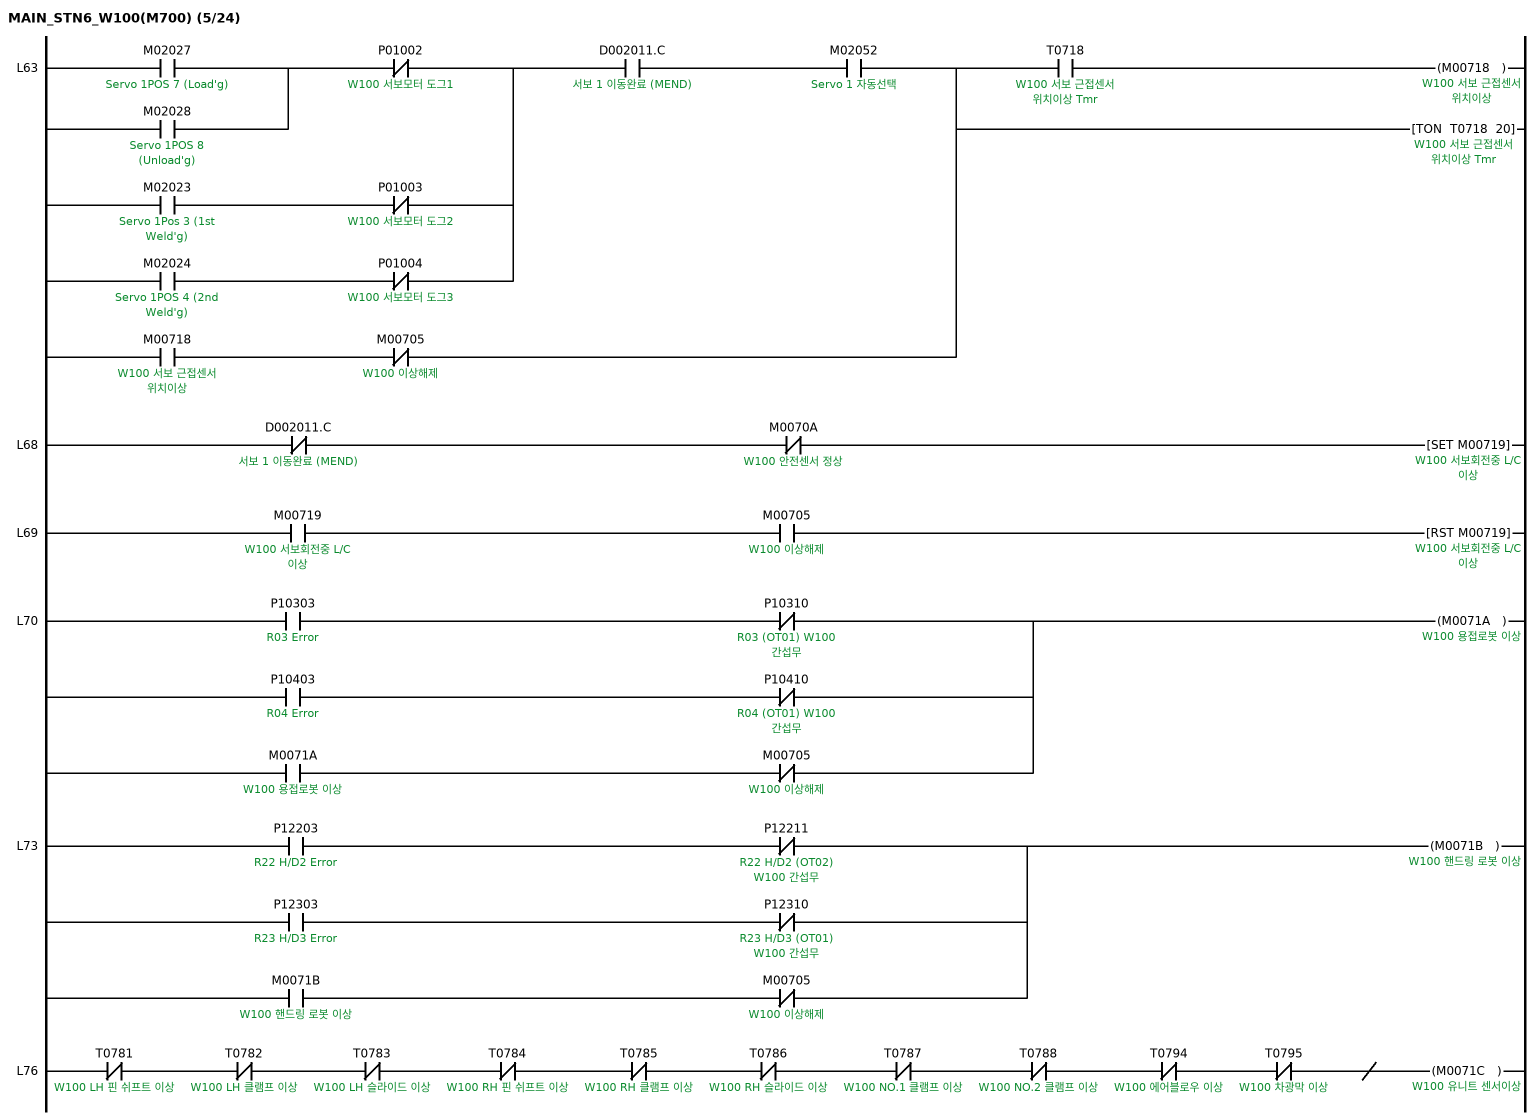
[picture p120: MAIN_STN6_W100(M700) rungs L63-L76]
; L63
LOAD      M02027	// Servo 1POS 7 (Load'g)
OR        M02028	// Servo 1POS 8 (Unload'g)
AND NOT   P01002	// W100 서보모터 도그1
LOAD      M02023	// Servo 1Pos 3 (1st Weld'g)
AND NOT   P01003	// W100 서보모터 도그2
OR LOAD
LOAD      M02024	// Servo 1POS 4 (2nd Weld'g)
AND NOT   P01004	// W100 서보모터 도그3
OR LOAD
AND       D002011.C	// 서보 1 이동완료 (MEND)
AND       M02052	// Servo 1 자동선택
LOAD      M00718	// W100 서보 근접센서 위치이상
AND NOT   M00705	// W100 이상해제
OR LOAD
MPUSH
AND       T0718	// W100 서보 근접센서 위치이상 Tmr
OUT       M00718	// W100 서보 근접센서 위치이상
MPOP
TON       T0718 20	// W100 서보 근접센서 위치이상 Tmr
; L68
LOAD NOT  D002011.C	// 서보 1 이동완료 (MEND)
AND NOT   M0070A	// W100 안전센서 정상
SET       M00719	// W100 서보회전중 L/C 이상
; L69
LOAD      M00719	// W100 서보회전중 L/C 이상
AND       M00705	// W100 이상해제
RST       M00719	// W100 서보회전중 L/C 이상
; L70
LOAD      P10303	// R03 Error
AND NOT   P10310	// R03 (OT01) W100 간섭무
LOAD      P10403	// R04 Error
AND NOT   P10410	// R04 (OT01) W100 간섭무
OR LOAD
LOAD      M0071A	// W100 용접로봇 이상
AND NOT   M00705	// W100 이상해제
OR LOAD
OUT       M0071A	// W100 용접로봇 이상
; L73
LOAD      P12203	// R22 H/D2 Error
AND NOT   P12211	// R22 H/D2 (OT02) W100 간섭무
LOAD      P12303	// R23 H/D3 Error
AND NOT   P12310	// R23 H/D3 (OT01) W100 간섭무
OR LOAD
LOAD      M0071B	// W100 핸드링 로봇 이상
AND NOT   M00705	// W100 이상해제
OR LOAD
OUT       M0071B	// W100 핸드링 로봇 이상
; L76
LOAD NOT  T0781	// W100 LH 핀 쉬프트 이상
AND NOT   T0782	// W100 LH 클램프 이상
AND NOT   T0783	// W100 LH 슬라이드 이상
AND NOT   T0784	// W100 RH 핀 쉬프트 이상
AND NOT   T0785	// W100 RH 클램프 이상
AND NOT   T0786	// W100 RH 슬라이드 이상
AND NOT   T0787	// W100 NO.1 클램프 이상
AND NOT   T0788	// W100 NO.2 클램프 이상
AND NOT   T0794	// W100 에어블로우 이상
AND NOT   T0795	// W100 차광막 이상
NOT
OUT       M0071C	// W100 유니트 센서이상

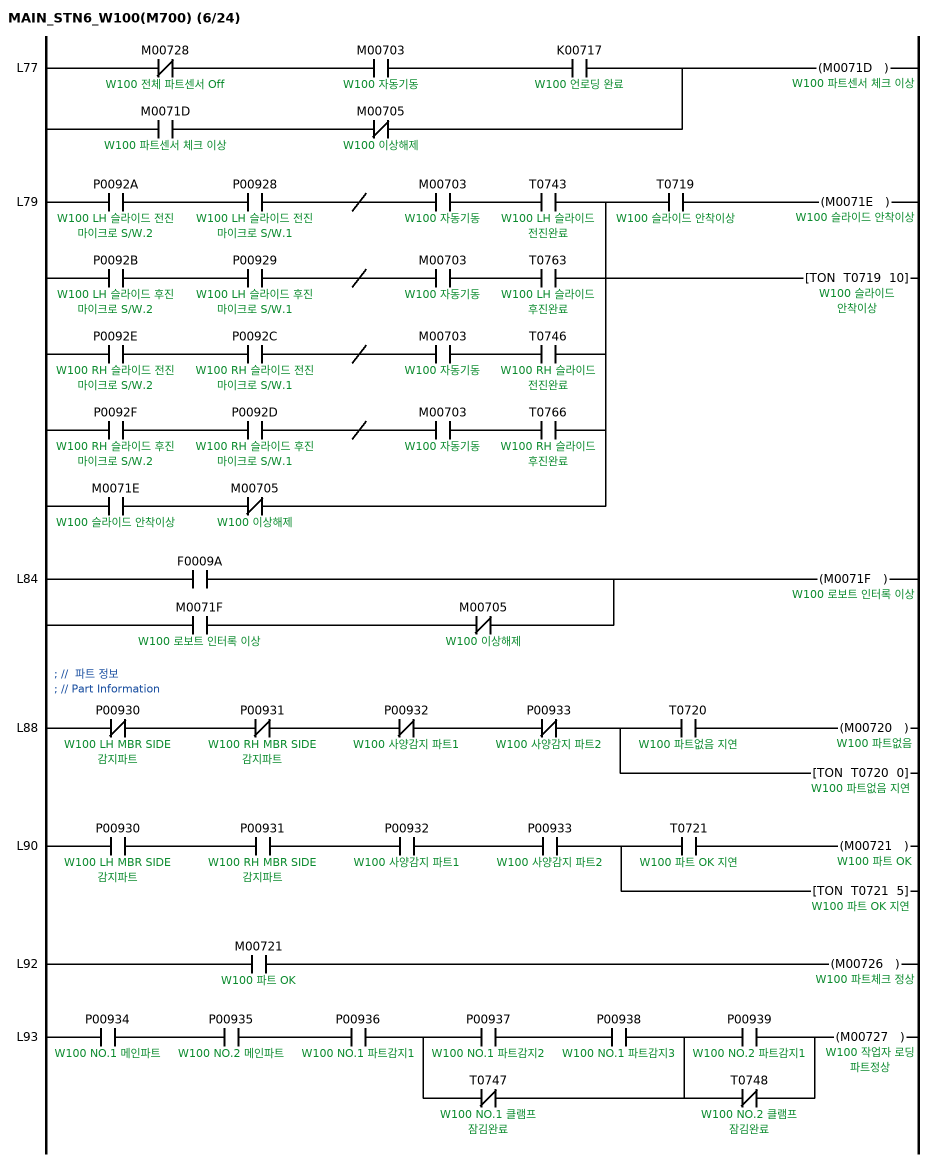
; L77
LOAD NOT  M00728	// W100 전체 파트센서 Off
AND       M00703	// W100 자동기동
AND       K00717	// W100 언로딩 완료
LOAD      M0071D	// W100 파트센서 체크 이상
AND NOT   M00705	// W100 이상해제
OR LOAD
OUT       M0071D	// W100 파트센서 체크 이상
; L79
LOAD      P0092A	// W100 LH 슬라이드 전진 마이크로 S/W.2
AND       P00928	// W100 LH 슬라이드 전진 마이크로 S/W.1
NOT
AND       M00703	// W100 자동기동
AND       T0743	// W100 LH 슬라이드 전진완료
LOAD      P0092B	// W100 LH 슬라이드 후진 마이크로 S/W.2
AND       P00929	// W100 LH 슬라이드 후진 마이크로 S/W.1
NOT
AND       M00703	// W100 자동기동
AND       T0763	// W100 LH 슬라이드 후진완료
OR LOAD
LOAD      P0092E	// W100 RH 슬라이드 전진 마이크로 S/W.2
AND       P0092C	// W100 RH 슬라이드 전진 마이크로 S/W.1
NOT
AND       M00703	// W100 자동기동
AND       T0746	// W100 RH 슬라이드 전진완료
OR LOAD
LOAD      P0092F	// W100 RH 슬라이드 후진 마이크로 S/W.2
AND       P0092D	// W100 RH 슬라이드 후진 마이크로 S/W.1
NOT
AND       M00703	// W100 자동기동
AND       T0766	// W100 RH 슬라이드 후진완료
OR LOAD
LOAD      M0071E	// W100 슬라이드 안착이상
AND NOT   M00705	// W100 이상해제
OR LOAD
MPUSH
AND       T0719	// W100 슬라이드 안착이상
OUT       M0071E	// W100 슬라이드 안착이상
MPOP
TON       T0719 10	// W100 슬라이드 안착이상
; L84
LOAD      F0009A
LOAD      M0071F	// W100 로보트 인터록 이상
AND NOT   M00705	// W100 이상해제
OR LOAD
OUT       M0071F	// W100 로보트 인터록 이상
//   //  파트 정보
//   // Part Information
; L88
LOAD NOT  P00930	// W100 LH MBR SIDE 감지파트
AND NOT   P00931	// W100 RH MBR SIDE 감지파트
AND NOT   P00932	// W100 사양감지 파트1
AND NOT   P00933	// W100 사양감지 파트2
MPUSH
AND       T0720	// W100 파트없음 지연
OUT       M00720	// W100 파트없음
MPOP
TON       T0720 0	// W100 파트없음 지연
; L90
LOAD      P00930	// W100 LH MBR SIDE 감지파트
AND       P00931	// W100 RH MBR SIDE 감지파트
AND       P00932	// W100 사양감지 파트1
AND       P00933	// W100 사양감지 파트2
MPUSH
AND       T0721	// W100 파트 OK 지연
OUT       M00721	// W100 파트 OK
MPOP
TON       T0721 5	// W100 파트 OK 지연
; L92
LOAD      M00721	// W100 파트 OK
OUT       M00726	// W100 파트체크 정상
; L93
LOAD      P00934	// W100 NO.1 메인파트
AND       P00935	// W100 NO.2 메인파트
AND       P00936	// W100 NO.1 파트감지1
LOAD      P00937	// W100 NO.1 파트감지2
AND       P00938	// W100 NO.1 파트감지3
OR NOT    T0747	// W100 NO.1 클램프 잠김완료
AND LOAD
LOAD      P00939	// W100 NO.2 파트감지1
OR NOT    T0748	// W100 NO.2 클램프 잠김완료
AND LOAD
OUT       M00727	// W100 작업자 로딩 파트정상

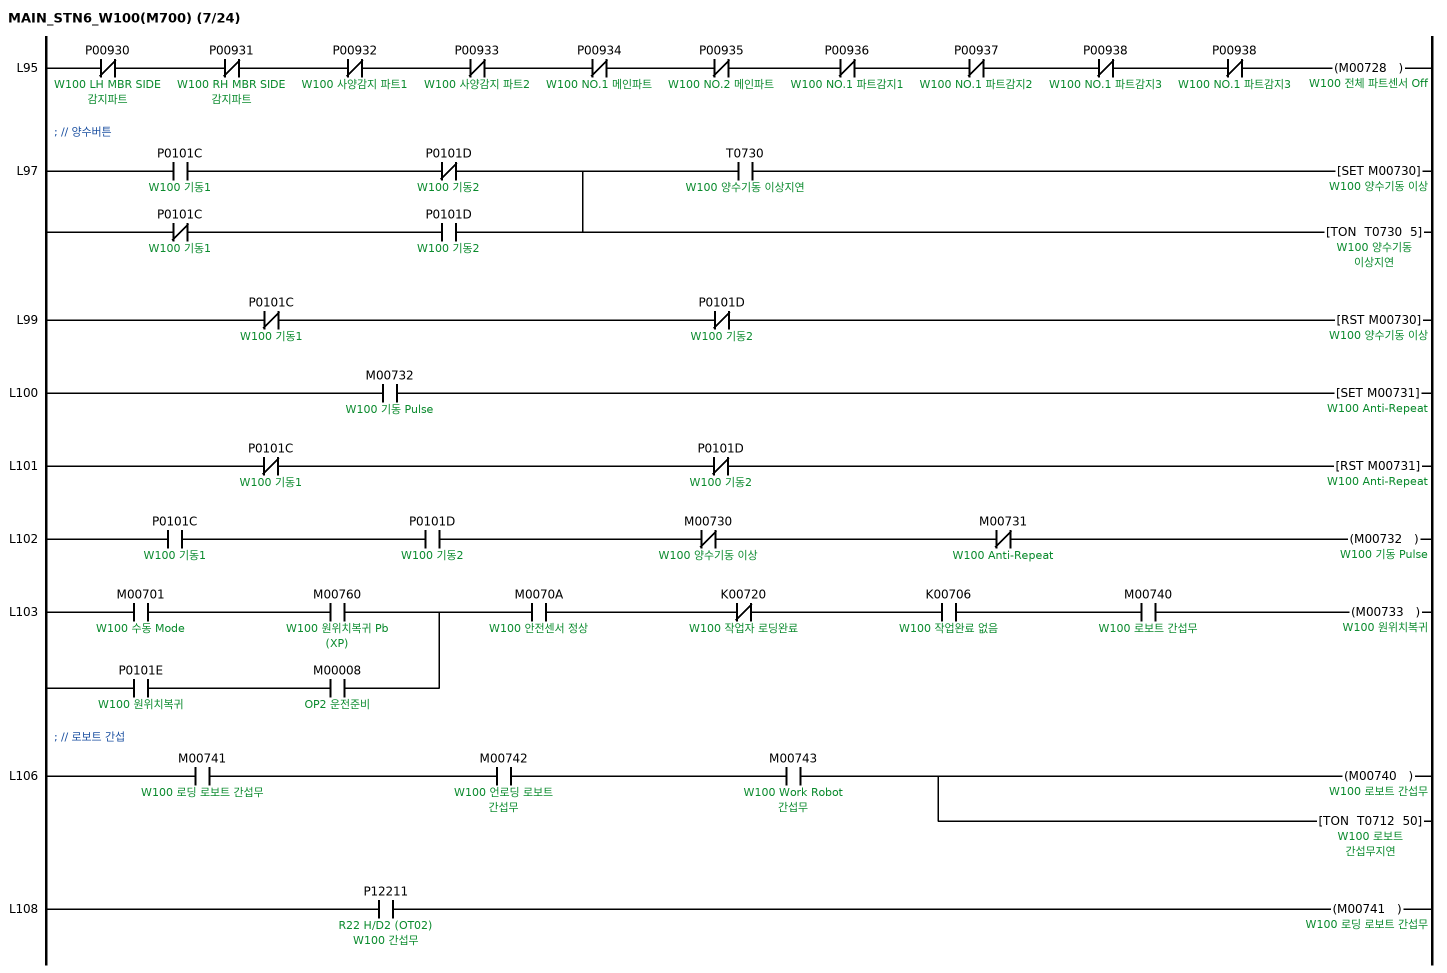
; L95
LOAD NOT  P00930	// W100 LH MBR SIDE 감지파트
AND NOT   P00931	// W100 RH MBR SIDE 감지파트
AND NOT   P00932	// W100 사양감지 파트1
AND NOT   P00933	// W100 사양감지 파트2
AND NOT   P00934	// W100 NO.1 메인파트
AND NOT   P00935	// W100 NO.2 메인파트
AND NOT   P00936	// W100 NO.1 파트감지1
AND NOT   P00937	// W100 NO.1 파트감지2
AND NOT   P00938	// W100 NO.1 파트감지3
AND NOT   P00938	// W100 NO.1 파트감지3
OUT       M00728	// W100 전체 파트센서 Off
//   // 양수버튼
; L97
LOAD      P0101C	// W100 기동1
AND NOT   P0101D	// W100 기동2
LOAD NOT  P0101C	// W100 기동1
AND       P0101D	// W100 기동2
OR LOAD
MPUSH
AND       T0730	// W100 양수기동 이상지연
SET       M00730	// W100 양수기동 이상
MPOP
TON       T0730 5	// W100 양수기동 이상지연
; L99
LOAD NOT  P0101C	// W100 기동1
AND NOT   P0101D	// W100 기동2
RST       M00730	// W100 양수기동 이상
; L100
LOAD      M00732	// W100 기동 Pulse
SET       M00731	// W100 Anti-Repeat
; L101
LOAD NOT  P0101C	// W100 기동1
AND NOT   P0101D	// W100 기동2
RST       M00731	// W100 Anti-Repeat
; L102
LOAD      P0101C	// W100 기동1
AND       P0101D	// W100 기동2
AND NOT   M00730	// W100 양수기동 이상
AND NOT   M00731	// W100 Anti-Repeat
OUT       M00732	// W100 기동 Pulse
; L103
LOAD      M00701	// W100 수동 Mode
AND       M00760	// W100 원위치복귀 Pb (XP)
LOAD      P0101E	// W100 원위치복귀
AND       M00008	// OP2 운전준비
OR LOAD
AND       M0070A	// W100 안전센서 정상
AND NOT   K00720	// W100 작업자 로딩완료
AND       K00706	// W100 작업완료 없음
AND       M00740	// W100 로보트 간섭무
OUT       M00733	// W100 원위치복귀
//   // 로보트 간섭
; L106
LOAD      M00741	// W100 로딩 로보트 간섭무
AND       M00742	// W100 언로딩 로보트 간섭무
AND       M00743	// W100 Work Robot 간섭무
OUT       M00740	// W100 로보트 간섭무
TON       T0712 50	// W100 로보트 간섭무지연
; L108
LOAD      P12211	// R22 H/D2 (OT02) W100 간섭무
OUT       M00741	// W100 로딩 로보트 간섭무

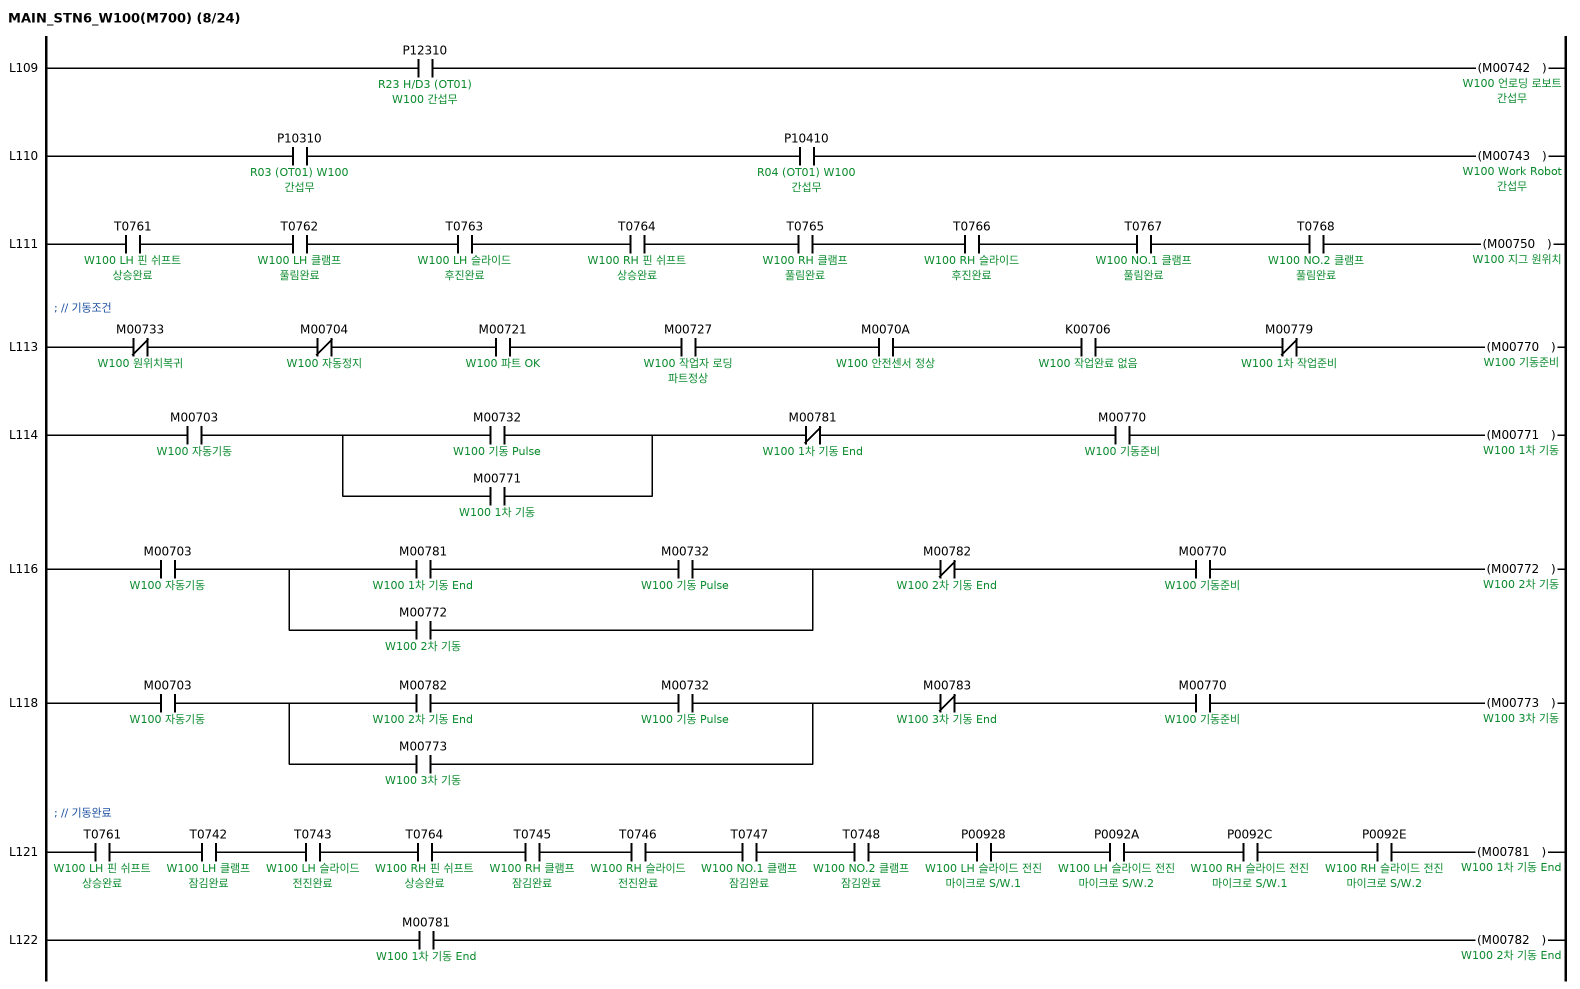
; L109
LOAD      P12310	// R23 H/D3 (OT01) W100 간섭무
OUT       M00742	// W100 언로딩 로보트 간섭무
; L110
LOAD      P10310	// R03 (OT01) W100 간섭무
AND       P10410	// R04 (OT01) W100 간섭무
OUT       M00743	// W100 Work Robot 간섭무
; L111
LOAD      T0761	// W100 LH 핀 쉬프트 상승완료
AND       T0762	// W100 LH 클램프 풀림완료
AND       T0763	// W100 LH 슬라이드 후진완료
AND       T0764	// W100 RH 핀 쉬프트 상승완료
AND       T0765	// W100 RH 클램프 풀림완료
AND       T0766	// W100 RH 슬라이드 후진완료
AND       T0767	// W100 NO.1 클램프 풀림완료
AND       T0768	// W100 NO.2 클램프 풀림완료
OUT       M00750	// W100 지그 원위치
//   // 기동조건
; L113
LOAD NOT  M00733	// W100 원위치복귀
AND NOT   M00704	// W100 자동정지
AND       M00721	// W100 파트 OK
AND       M00727	// W100 작업자 로딩 파트정상
AND       M0070A	// W100 안전센서 정상
AND       K00706	// W100 작업완료 없음
AND NOT   M00779	// W100 1차 작업준비
OUT       M00770	// W100 기동준비
; L114
LOAD      M00703	// W100 자동기동
LOAD      M00732	// W100 기동 Pulse
OR        M00771	// W100 1차 기동
AND LOAD
AND NOT   M00781	// W100 1차 기동 End
AND       M00770	// W100 기동준비
OUT       M00771	// W100 1차 기동
; L116
LOAD      M00703	// W100 자동기동
LOAD      M00781	// W100 1차 기동 End
AND       M00732	// W100 기동 Pulse
OR        M00772	// W100 2차 기동
AND LOAD
AND NOT   M00782	// W100 2차 기동 End
AND       M00770	// W100 기동준비
OUT       M00772	// W100 2차 기동
; L118
LOAD      M00703	// W100 자동기동
LOAD      M00782	// W100 2차 기동 End
AND       M00732	// W100 기동 Pulse
OR        M00773	// W100 3차 기동
AND LOAD
AND NOT   M00783	// W100 3차 기동 End
AND       M00770	// W100 기동준비
OUT       M00773	// W100 3차 기동
//   // 기동완료
; L121
LOAD      T0761	// W100 LH 핀 쉬프트 상승완료
AND       T0742	// W100 LH 클램프 잠김완료
AND       T0743	// W100 LH 슬라이드 전진완료
AND       T0764	// W100 RH 핀 쉬프트 상승완료
AND       T0745	// W100 RH 클램프 잠김완료
AND       T0746	// W100 RH 슬라이드 전진완료
AND       T0747	// W100 NO.1 클램프 잠김완료
AND       T0748	// W100 NO.2 클램프 잠김완료
AND       P00928	// W100 LH 슬라이드 전진 마이크로 S/W.1
AND       P0092A	// W100 LH 슬라이드 전진 마이크로 S/W.2
AND       P0092C	// W100 RH 슬라이드 전진 마이크로 S/W.1
AND       P0092E	// W100 RH 슬라이드 전진 마이크로 S/W.2
OUT       M00781	// W100 1차 기동 End
; L122
LOAD      M00781	// W100 1차 기동 End
OUT       M00782	// W100 2차 기동 End

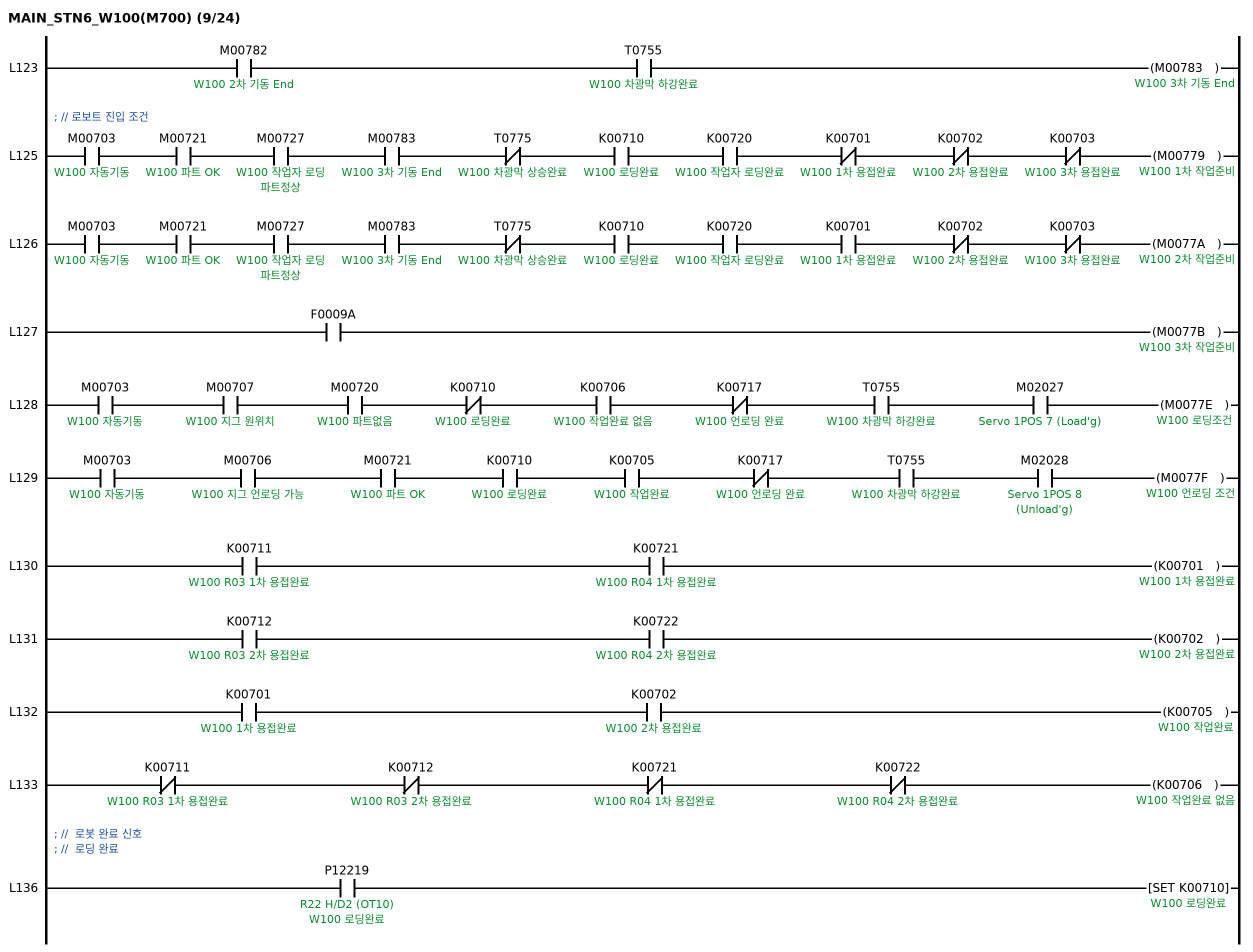
; L123
LOAD      M00782	// W100 2차 기동 End
AND       T0755	// W100 차광막 하강완료
OUT       M00783	// W100 3차 기동 End
//   // 로보트 진입 조건
; L125
LOAD      M00703	// W100 자동기동
AND       M00721	// W100 파트 OK
AND       M00727	// W100 작업자 로딩 파트정상
AND       M00783	// W100 3차 기동 End
AND NOT   T0775	// W100 차광막 상승완료
AND       K00710	// W100 로딩완료
AND       K00720	// W100 작업자 로딩완료
AND NOT   K00701	// W100 1차 용접완료
AND NOT   K00702	// W100 2차 용접완료
AND NOT   K00703	// W100 3차 용접완료
OUT       M00779	// W100 1차 작업준비
; L126
LOAD      M00703	// W100 자동기동
AND       M00721	// W100 파트 OK
AND       M00727	// W100 작업자 로딩 파트정상
AND       M00783	// W100 3차 기동 End
AND NOT   T0775	// W100 차광막 상승완료
AND       K00710	// W100 로딩완료
AND       K00720	// W100 작업자 로딩완료
AND       K00701	// W100 1차 용접완료
AND NOT   K00702	// W100 2차 용접완료
AND NOT   K00703	// W100 3차 용접완료
OUT       M0077A	// W100 2차 작업준비
; L127
LOAD      F0009A
OUT       M0077B	// W100 3차 작업준비
; L128
LOAD      M00703	// W100 자동기동
AND       M00707	// W100 지그 원위치
AND       M00720	// W100 파트없음
AND NOT   K00710	// W100 로딩완료
AND       K00706	// W100 작업완료 없음
AND NOT   K00717	// W100 언로딩 완료
AND       T0755	// W100 차광막 하강완료
AND       M02027	// Servo 1POS 7 (Load'g)
OUT       M0077E	// W100 로딩조건
; L129
LOAD      M00703	// W100 자동기동
AND       M00706	// W100 지그 언로딩 가능
AND       M00721	// W100 파트 OK
AND       K00710	// W100 로딩완료
AND       K00705	// W100 작업완료
AND NOT   K00717	// W100 언로딩 완료
AND       T0755	// W100 차광막 하강완료
AND       M02028	// Servo 1POS 8 (Unload'g)
OUT       M0077F	// W100 언로딩 조건
; L130
LOAD      K00711	// W100 R03 1차 용접완료
AND       K00721	// W100 R04 1차 용접완료
OUT       K00701	// W100 1차 용접완료
; L131
LOAD      K00712	// W100 R03 2차 용접완료
AND       K00722	// W100 R04 2차 용접완료
OUT       K00702	// W100 2차 용접완료
; L132
LOAD      K00701	// W100 1차 용접완료
AND       K00702	// W100 2차 용접완료
OUT       K00705	// W100 작업완료
; L133
LOAD NOT  K00711	// W100 R03 1차 용접완료
AND NOT   K00712	// W100 R03 2차 용접완료
AND NOT   K00721	// W100 R04 1차 용접완료
AND NOT   K00722	// W100 R04 2차 용접완료
OUT       K00706	// W100 작업완료 없음
//   //  로봇 완료 신호
//   //  로딩 완료
; L136
LOAD      P12219	// R22 H/D2 (OT10) W100 로딩완료
SET       K00710	// W100 로딩완료

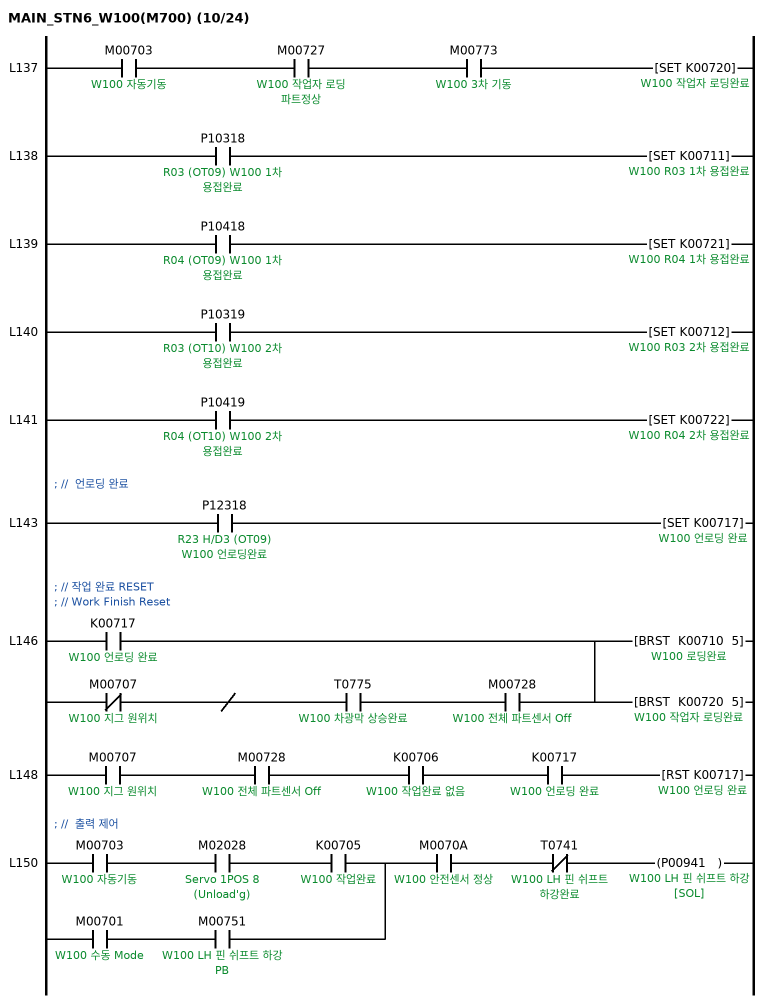
; L137
LOAD      M00703	// W100 자동기동
AND       M00727	// W100 작업자 로딩 파트정상
AND       M00773	// W100 3차 기동
SET       K00720	// W100 작업자 로딩완료
; L138
LOAD      P10318	// R03 (OT09) W100 1차 용접완료
SET       K00711	// W100 R03 1차 용접완료
; L139
LOAD      P10418	// R04 (OT09) W100 1차 용접완료
SET       K00721	// W100 R04 1차 용접완료
; L140
LOAD      P10319	// R03 (OT10) W100 2차 용접완료
SET       K00712	// W100 R03 2차 용접완료
; L141
LOAD      P10419	// R04 (OT10) W100 2차 용접완료
SET       K00722	// W100 R04 2차 용접완료
//   //  언로딩 완료
; L143
LOAD      P12318	// R23 H/D3 (OT09) W100 언로딩완료
SET       K00717	// W100 언로딩 완료
//     // 작업 완료 RESET
//   // Work Finish Reset
; L146
LOAD      K00717	// W100 언로딩 완료
LOAD NOT  M00707	// W100 지그 원위치
NOT
AND       T0775	// W100 차광막 상승완료
AND       M00728	// W100 전체 파트센서 Off
OR LOAD
BRST      K00710 5	// W100 로딩완료
BRST      K00720 5	// W100 작업자 로딩완료
; L148
LOAD      M00707	// W100 지그 원위치
AND       M00728	// W100 전체 파트센서 Off
AND       K00706	// W100 작업완료 없음
AND       K00717	// W100 언로딩 완료
RST       K00717	// W100 언로딩 완료
//     //  출력 제어
; L150
LOAD      M00703	// W100 자동기동
AND       M02028	// Servo 1POS 8 (Unload'g)
AND       K00705	// W100 작업완료
LOAD      M00701	// W100 수동 Mode
AND       M00751	// W100 LH 핀 쉬프트 하강 PB
OR LOAD
AND       M0070A	// W100 안전센서 정상
AND NOT   T0741	// W100 LH 핀 쉬프트 하강완료
OUT       P00941	// W100 LH 핀 쉬프트 하강 [SOL]

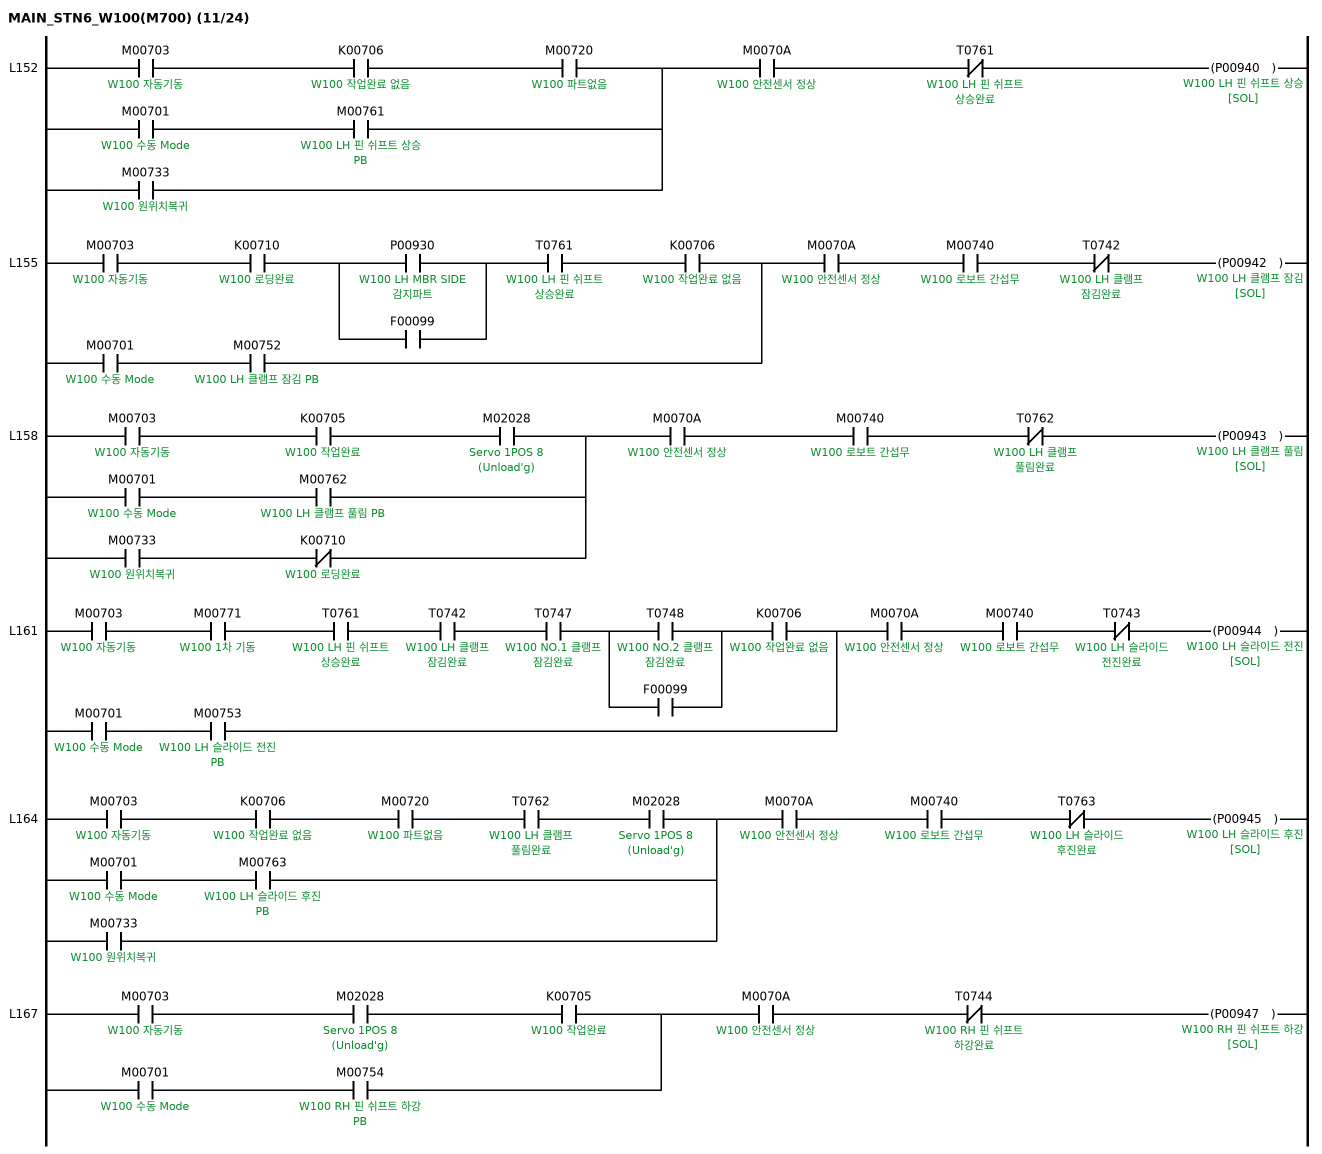
; L152
LOAD      M00703	// W100 자동기동
AND       K00706	// W100 작업완료 없음
AND       M00720	// W100 파트없음
LOAD      M00701	// W100 수동 Mode
AND       M00761	// W100 LH 핀 쉬프트 상승 PB
OR LOAD
OR        M00733	// W100 원위치복귀
AND       M0070A	// W100 안전센서 정상
AND NOT   T0761	// W100 LH 핀 쉬프트 상승완료
OUT       P00940	// W100 LH 핀 쉬프트 상승 [SOL]
; L155
LOAD      M00703	// W100 자동기동
AND       K00710	// W100 로딩완료
LOAD      P00930	// W100 LH MBR SIDE 감지파트
OR        F00099
AND LOAD
AND       T0761	// W100 LH 핀 쉬프트 상승완료
AND       K00706	// W100 작업완료 없음
LOAD      M00701	// W100 수동 Mode
AND       M00752	// W100 LH 클램프 잠김 PB
OR LOAD
AND       M0070A	// W100 안전센서 정상
AND       M00740	// W100 로보트 간섭무
AND NOT   T0742	// W100 LH 클램프 잠김완료
OUT       P00942	// W100 LH 클램프 잠김 [SOL]
; L158
LOAD      M00703	// W100 자동기동
AND       K00705	// W100 작업완료
AND       M02028	// Servo 1POS 8 (Unload'g)
LOAD      M00701	// W100 수동 Mode
AND       M00762	// W100 LH 클램프 풀림 PB
OR LOAD
LOAD      M00733	// W100 원위치복귀
AND NOT   K00710	// W100 로딩완료
OR LOAD
AND       M0070A	// W100 안전센서 정상
AND       M00740	// W100 로보트 간섭무
AND NOT   T0762	// W100 LH 클램프 풀림완료
OUT       P00943	// W100 LH 클램프 풀림 [SOL]
; L161
LOAD      M00703	// W100 자동기동
AND       M00771	// W100 1차 기동
AND       T0761	// W100 LH 핀 쉬프트 상승완료
AND       T0742	// W100 LH 클램프 잠김완료
AND       T0747	// W100 NO.1 클램프 잠김완료
LOAD      T0748	// W100 NO.2 클램프 잠김완료
OR        F00099
AND LOAD
AND       K00706	// W100 작업완료 없음
LOAD      M00701	// W100 수동 Mode
AND       M00753	// W100 LH 슬라이드 전진 PB
OR LOAD
AND       M0070A	// W100 안전센서 정상
AND       M00740	// W100 로보트 간섭무
AND NOT   T0743	// W100 LH 슬라이드 전진완료
OUT       P00944	// W100 LH 슬라이드 전진 [SOL]
; L164
LOAD      M00703	// W100 자동기동
AND       K00706	// W100 작업완료 없음
AND       M00720	// W100 파트없음
AND       T0762	// W100 LH 클램프 풀림완료
AND       M02028	// Servo 1POS 8 (Unload'g)
LOAD      M00701	// W100 수동 Mode
AND       M00763	// W100 LH 슬라이드 후진 PB
OR LOAD
OR        M00733	// W100 원위치복귀
AND       M0070A	// W100 안전센서 정상
AND       M00740	// W100 로보트 간섭무
AND NOT   T0763	// W100 LH 슬라이드 후진완료
OUT       P00945	// W100 LH 슬라이드 후진 [SOL]
; L167
LOAD      M00703	// W100 자동기동
AND       M02028	// Servo 1POS 8 (Unload'g)
AND       K00705	// W100 작업완료
LOAD      M00701	// W100 수동 Mode
AND       M00754	// W100 RH 핀 쉬프트 하강 PB
OR LOAD
AND       M0070A	// W100 안전센서 정상
AND NOT   T0744	// W100 RH 핀 쉬프트 하강완료
OUT       P00947	// W100 RH 핀 쉬프트 하강 [SOL]

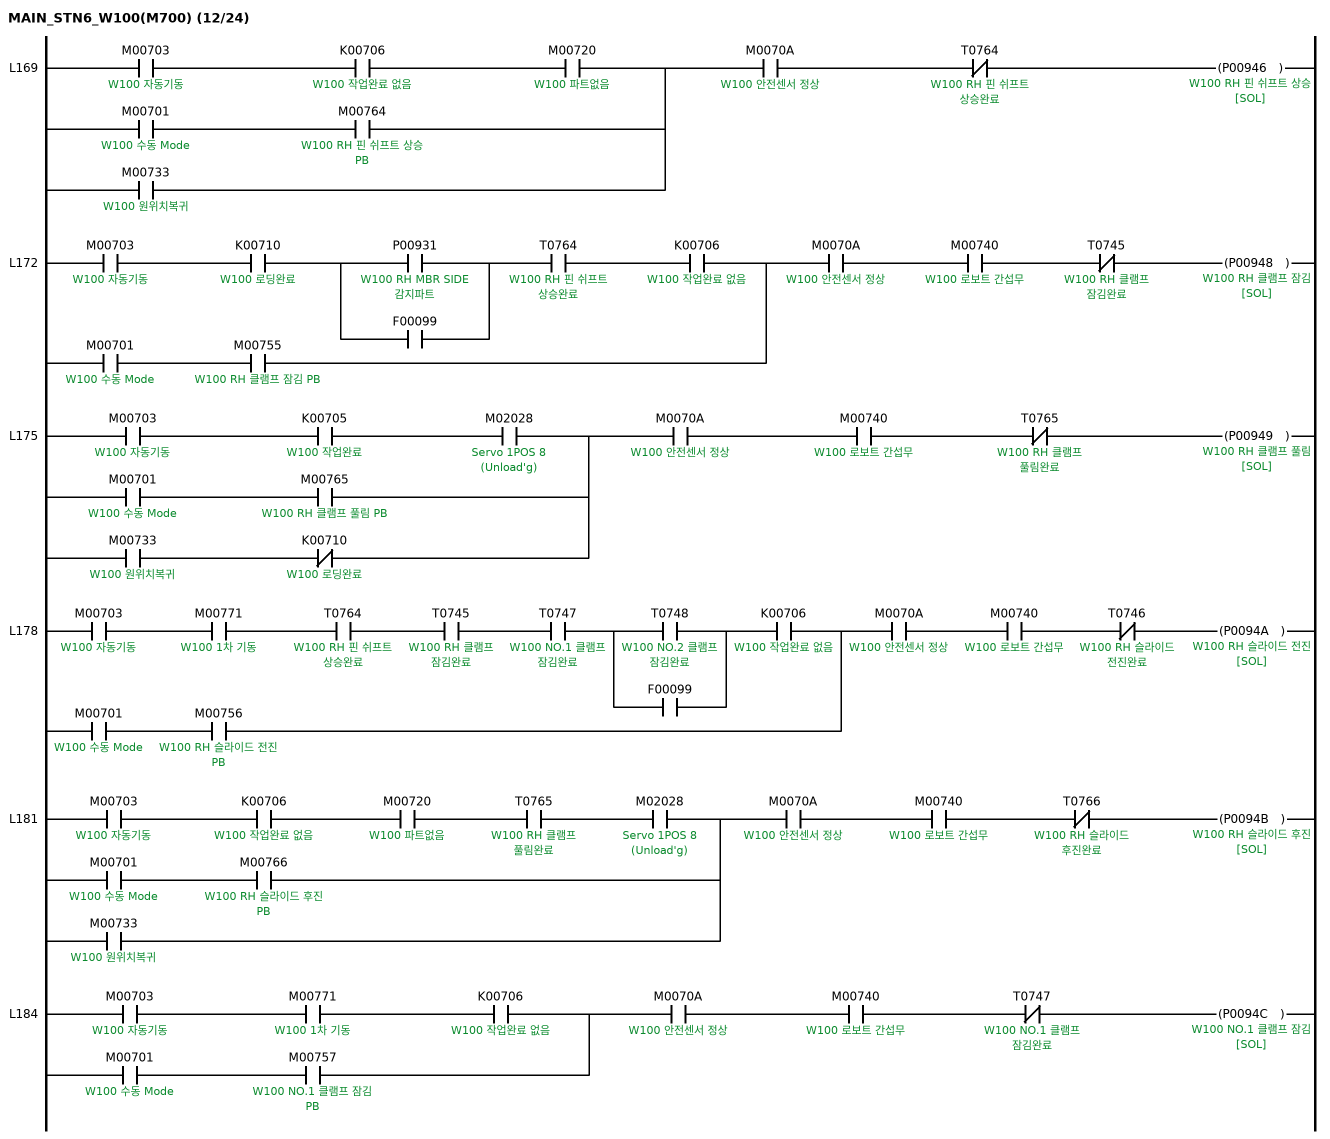
; L169
LOAD      M00703	// W100 자동기동
AND       K00706	// W100 작업완료 없음
AND       M00720	// W100 파트없음
LOAD      M00701	// W100 수동 Mode
AND       M00764	// W100 RH 핀 쉬프트 상승 PB
OR LOAD
OR        M00733	// W100 원위치복귀
AND       M0070A	// W100 안전센서 정상
AND NOT   T0764	// W100 RH 핀 쉬프트 상승완료
OUT       P00946	// W100 RH 핀 쉬프트 상승 [SOL]
; L172
LOAD      M00703	// W100 자동기동
AND       K00710	// W100 로딩완료
LOAD      P00931	// W100 RH MBR SIDE 감지파트
OR        F00099
AND LOAD
AND       T0764	// W100 RH 핀 쉬프트 상승완료
AND       K00706	// W100 작업완료 없음
LOAD      M00701	// W100 수동 Mode
AND       M00755	// W100 RH 클램프 잠김 PB
OR LOAD
AND       M0070A	// W100 안전센서 정상
AND       M00740	// W100 로보트 간섭무
AND NOT   T0745	// W100 RH 클램프 잠김완료
OUT       P00948	// W100 RH 클램프 잠김 [SOL]
; L175
LOAD      M00703	// W100 자동기동
AND       K00705	// W100 작업완료
AND       M02028	// Servo 1POS 8 (Unload'g)
LOAD      M00701	// W100 수동 Mode
AND       M00765	// W100 RH 클램프 풀림 PB
OR LOAD
LOAD      M00733	// W100 원위치복귀
AND NOT   K00710	// W100 로딩완료
OR LOAD
AND       M0070A	// W100 안전센서 정상
AND       M00740	// W100 로보트 간섭무
AND NOT   T0765	// W100 RH 클램프 풀림완료
OUT       P00949	// W100 RH 클램프 풀림 [SOL]
; L178
LOAD      M00703	// W100 자동기동
AND       M00771	// W100 1차 기동
AND       T0764	// W100 RH 핀 쉬프트 상승완료
AND       T0745	// W100 RH 클램프 잠김완료
AND       T0747	// W100 NO.1 클램프 잠김완료
LOAD      T0748	// W100 NO.2 클램프 잠김완료
OR        F00099
AND LOAD
AND       K00706	// W100 작업완료 없음
LOAD      M00701	// W100 수동 Mode
AND       M00756	// W100 RH 슬라이드 전진 PB
OR LOAD
AND       M0070A	// W100 안전센서 정상
AND       M00740	// W100 로보트 간섭무
AND NOT   T0746	// W100 RH 슬라이드 전진완료
OUT       P0094A	// W100 RH 슬라이드 전진 [SOL]
; L181
LOAD      M00703	// W100 자동기동
AND       K00706	// W100 작업완료 없음
AND       M00720	// W100 파트없음
AND       T0765	// W100 RH 클램프 풀림완료
AND       M02028	// Servo 1POS 8 (Unload'g)
LOAD      M00701	// W100 수동 Mode
AND       M00766	// W100 RH 슬라이드 후진 PB
OR LOAD
OR        M00733	// W100 원위치복귀
AND       M0070A	// W100 안전센서 정상
AND       M00740	// W100 로보트 간섭무
AND NOT   T0766	// W100 RH 슬라이드 후진완료
OUT       P0094B	// W100 RH 슬라이드 후진 [SOL]
; L184
LOAD      M00703	// W100 자동기동
AND       M00771	// W100 1차 기동
AND       K00706	// W100 작업완료 없음
LOAD      M00701	// W100 수동 Mode
AND       M00757	// W100 NO.1 클램프 잠김 PB
OR LOAD
AND       M0070A	// W100 안전센서 정상
AND       M00740	// W100 로보트 간섭무
AND NOT   T0747	// W100 NO.1 클램프 잠김완료
OUT       P0094C	// W100 NO.1 클램프 잠김 [SOL]

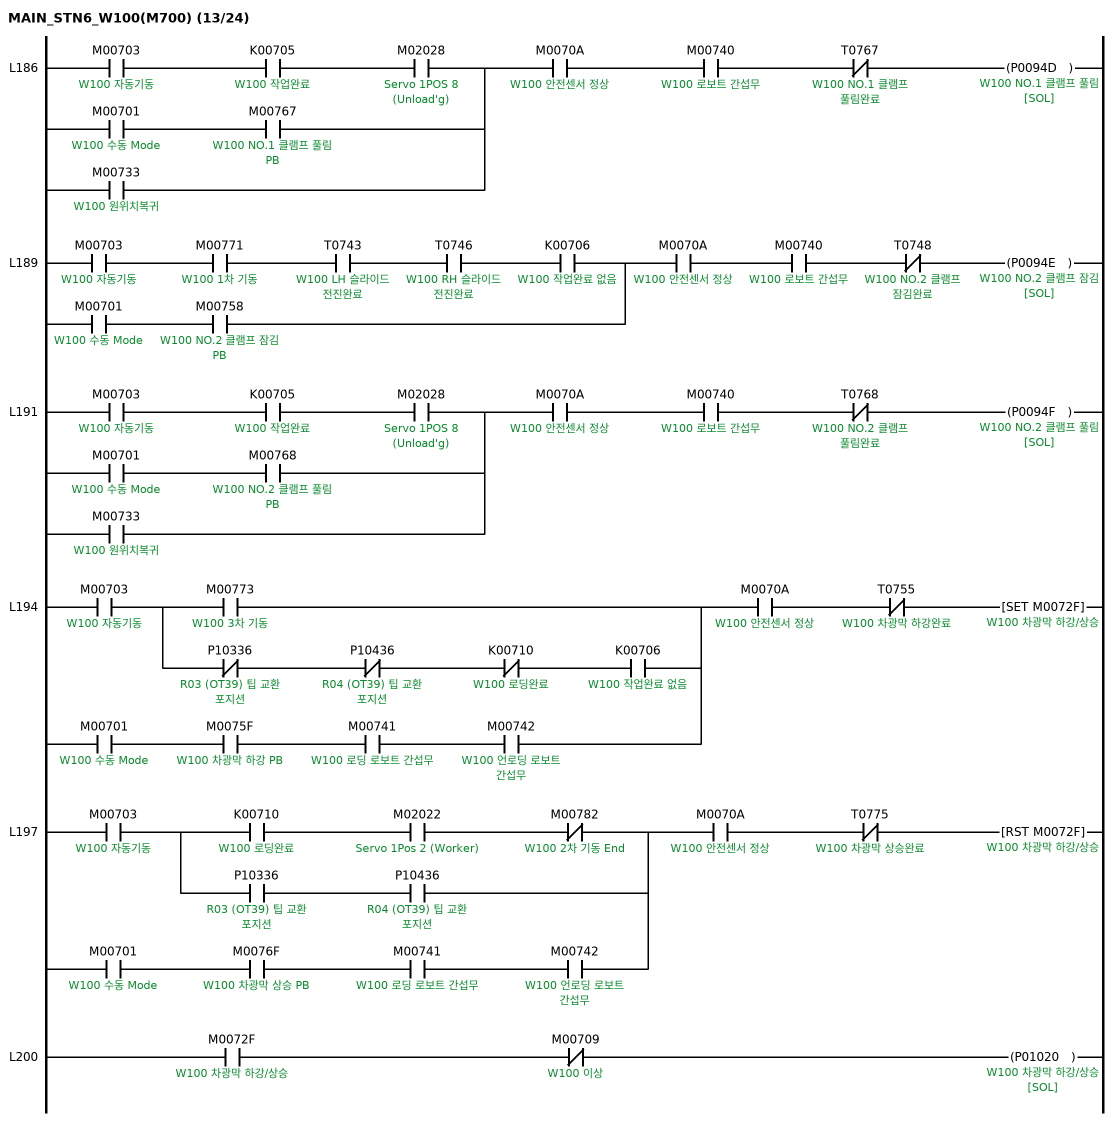
; L186
LOAD      M00703	// W100 자동기동
AND       K00705	// W100 작업완료
AND       M02028	// Servo 1POS 8 (Unload'g)
LOAD      M00701	// W100 수동 Mode
AND       M00767	// W100 NO.1 클램프 풀림 PB
OR LOAD
OR        M00733	// W100 원위치복귀
AND       M0070A	// W100 안전센서 정상
AND       M00740	// W100 로보트 간섭무
AND NOT   T0767	// W100 NO.1 클램프 풀림완료
OUT       P0094D	// W100 NO.1 클램프 풀림 [SOL]
; L189
LOAD      M00703	// W100 자동기동
AND       M00771	// W100 1차 기동
AND       T0743	// W100 LH 슬라이드 전진완료
AND       T0746	// W100 RH 슬라이드 전진완료
AND       K00706	// W100 작업완료 없음
LOAD      M00701	// W100 수동 Mode
AND       M00758	// W100 NO.2 클램프 잠김 PB
OR LOAD
AND       M0070A	// W100 안전센서 정상
AND       M00740	// W100 로보트 간섭무
AND NOT   T0748	// W100 NO.2 클램프 잠김완료
OUT       P0094E	// W100 NO.2 클램프 잠김 [SOL]
; L191
LOAD      M00703	// W100 자동기동
AND       K00705	// W100 작업완료
AND       M02028	// Servo 1POS 8 (Unload'g)
LOAD      M00701	// W100 수동 Mode
AND       M00768	// W100 NO.2 클램프 풀림 PB
OR LOAD
OR        M00733	// W100 원위치복귀
AND       M0070A	// W100 안전센서 정상
AND       M00740	// W100 로보트 간섭무
AND NOT   T0768	// W100 NO.2 클램프 풀림완료
OUT       P0094F	// W100 NO.2 클램프 풀림 [SOL]
; L194
LOAD      M00703	// W100 자동기동
LOAD      M00773	// W100 3차 기동
LOAD NOT  P10336	// R03 (OT39) 팁 교환 포지션
AND NOT   P10436	// R04 (OT39) 팁 교환 포지션
AND NOT   K00710	// W100 로딩완료
AND       K00706	// W100 작업완료 없음
OR LOAD
AND LOAD
LOAD      M00701	// W100 수동 Mode
AND       M0075F	// W100 차광막 하강 PB
AND       M00741	// W100 로딩 로보트 간섭무
AND       M00742	// W100 언로딩 로보트 간섭무
OR LOAD
AND       M0070A	// W100 안전센서 정상
AND NOT   T0755	// W100 차광막 하강완료
SET       M0072F	// W100 차광막 하강/상승
; L197
LOAD      M00703	// W100 자동기동
LOAD      K00710	// W100 로딩완료
AND       M02022	// Servo 1Pos 2 (Worker)
AND NOT   M00782	// W100 2차 기동 End
LOAD      P10336	// R03 (OT39) 팁 교환 포지션
AND       P10436	// R04 (OT39) 팁 교환 포지션
OR LOAD
AND LOAD
LOAD      M00701	// W100 수동 Mode
AND       M0076F	// W100 차광막 상승 PB
AND       M00741	// W100 로딩 로보트 간섭무
AND       M00742	// W100 언로딩 로보트 간섭무
OR LOAD
AND       M0070A	// W100 안전센서 정상
AND NOT   T0775	// W100 차광막 상승완료
RST       M0072F	// W100 차광막 하강/상승
; L200
LOAD      M0072F	// W100 차광막 하강/상승
AND NOT   M00709	// W100 이상
OUT       P01020	// W100 차광막 하강/상승 [SOL]

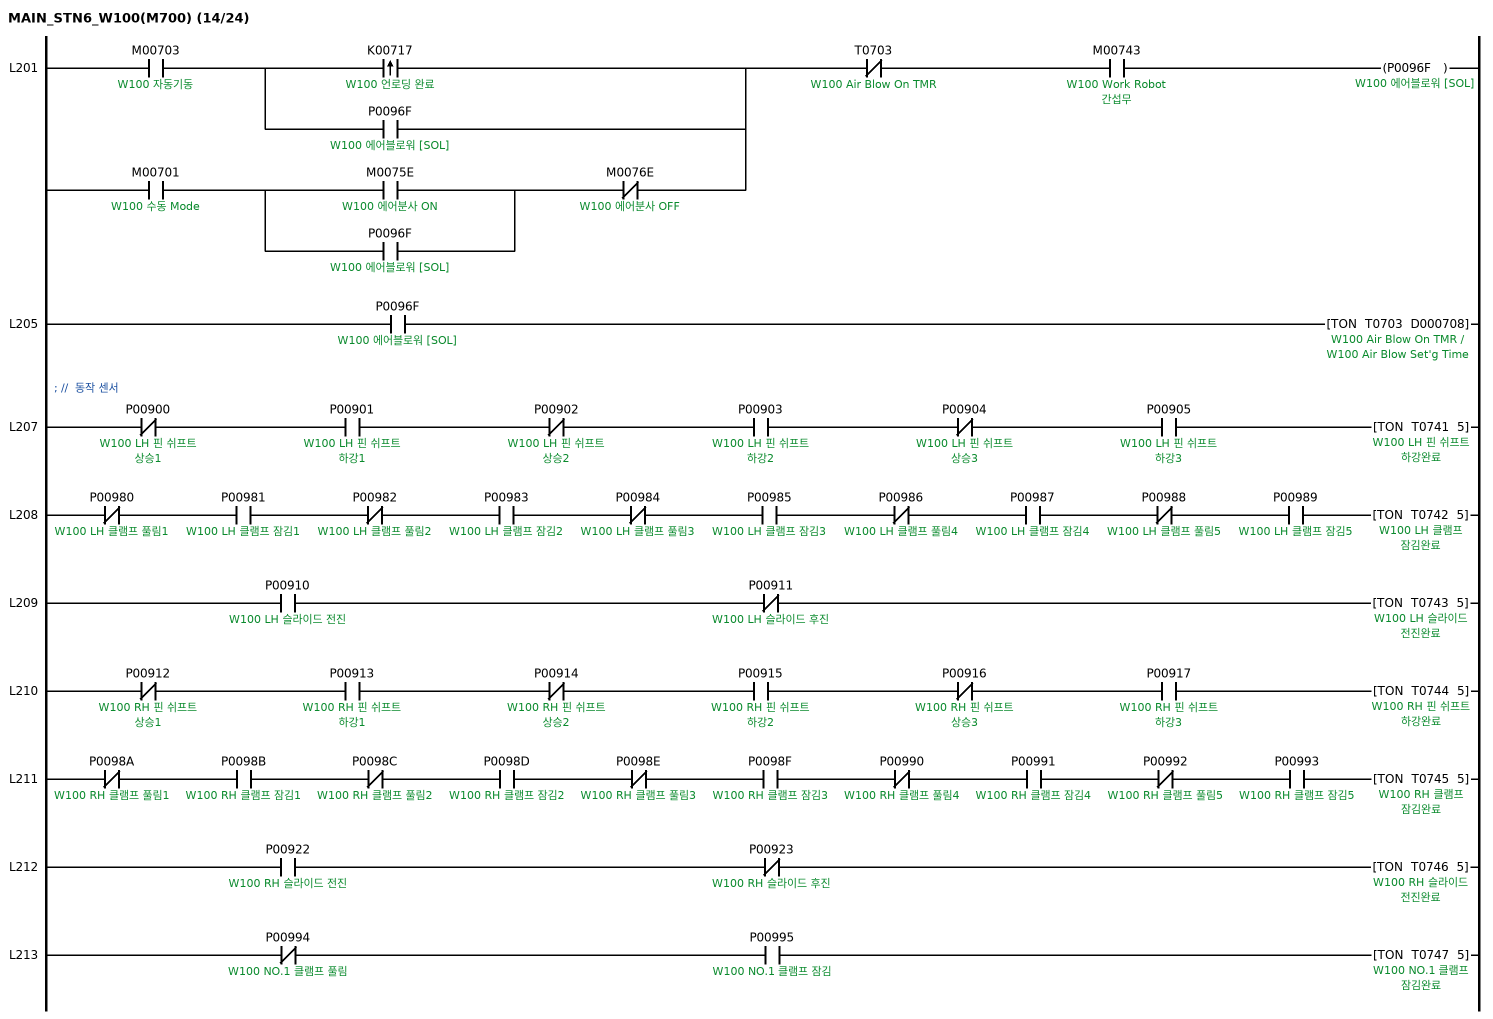
; L201
LOAD      M00703	// W100 자동기동
LOADP     K00717	// W100 언로딩 완료
OR        P0096F	// W100 에어블로워 [SOL]
AND LOAD
LOAD      M00701	// W100 수동 Mode
LOAD      M0075E	// W100 에어분사 ON
OR        P0096F	// W100 에어블로워 [SOL]
AND LOAD
AND NOT   M0076E	// W100 에어분사 OFF
OR LOAD
AND NOT   T0703	// W100 Air Blow On TMR
AND       M00743	// W100 Work Robot 간섭무
OUT       P0096F	// W100 에어블로워 [SOL]
; L205
LOAD      P0096F	// W100 에어블로워 [SOL]
TON       T0703 D000708	// W100 Air Blow On TMR / W100 Air Blow Set'g Time
//   //  동작 센서
; L207
LOAD NOT  P00900	// W100 LH 핀 쉬프트 상승1
AND       P00901	// W100 LH 핀 쉬프트 하강1
AND NOT   P00902	// W100 LH 핀 쉬프트 상승2
AND       P00903	// W100 LH 핀 쉬프트 하강2
AND NOT   P00904	// W100 LH 핀 쉬프트 상승3
AND       P00905	// W100 LH 핀 쉬프트 하강3
TON       T0741 5	// W100 LH 핀 쉬프트 하강완료
; L208
LOAD NOT  P00980	// W100 LH 클램프 풀림1
AND       P00981	// W100 LH 클램프 잠김1
AND NOT   P00982	// W100 LH 클램프 풀림2
AND       P00983	// W100 LH 클램프 잠김2
AND NOT   P00984	// W100 LH 클램프 풀림3
AND       P00985	// W100 LH 클램프 잠김3
AND NOT   P00986	// W100 LH 클램프 풀림4
AND       P00987	// W100 LH 클램프 잠김4
AND NOT   P00988	// W100 LH 클램프 풀림5
AND       P00989	// W100 LH 클램프 잠김5
TON       T0742 5	// W100 LH 클램프 잠김완료
; L209
LOAD      P00910	// W100 LH 슬라이드 전진
AND NOT   P00911	// W100 LH 슬라이드 후진
TON       T0743 5	// W100 LH 슬라이드 전진완료
; L210
LOAD NOT  P00912	// W100 RH 핀 쉬프트 상승1
AND       P00913	// W100 RH 핀 쉬프트 하강1
AND NOT   P00914	// W100 RH 핀 쉬프트 상승2
AND       P00915	// W100 RH 핀 쉬프트 하강2
AND NOT   P00916	// W100 RH 핀 쉬프트 상승3
AND       P00917	// W100 RH 핀 쉬프트 하강3
TON       T0744 5	// W100 RH 핀 쉬프트 하강완료
; L211
LOAD NOT  P0098A	// W100 RH 클램프 풀림1
AND       P0098B	// W100 RH 클램프 잠김1
AND NOT   P0098C	// W100 RH 클램프 풀림2
AND       P0098D	// W100 RH 클램프 잠김2
AND NOT   P0098E	// W100 RH 클램프 풀림3
AND       P0098F	// W100 RH 클램프 잠김3
AND NOT   P00990	// W100 RH 클램프 풀림4
AND       P00991	// W100 RH 클램프 잠김4
AND NOT   P00992	// W100 RH 클램프 풀림5
AND       P00993	// W100 RH 클램프 잠김5
TON       T0745 5	// W100 RH 클램프 잠김완료
; L212
LOAD      P00922	// W100 RH 슬라이드 전진
AND NOT   P00923	// W100 RH 슬라이드 후진
TON       T0746 5	// W100 RH 슬라이드 전진완료
; L213
LOAD NOT  P00994	// W100 NO.1 클램프 풀림
AND       P00995	// W100 NO.1 클램프 잠김
TON       T0747 5	// W100 NO.1 클램프 잠김완료

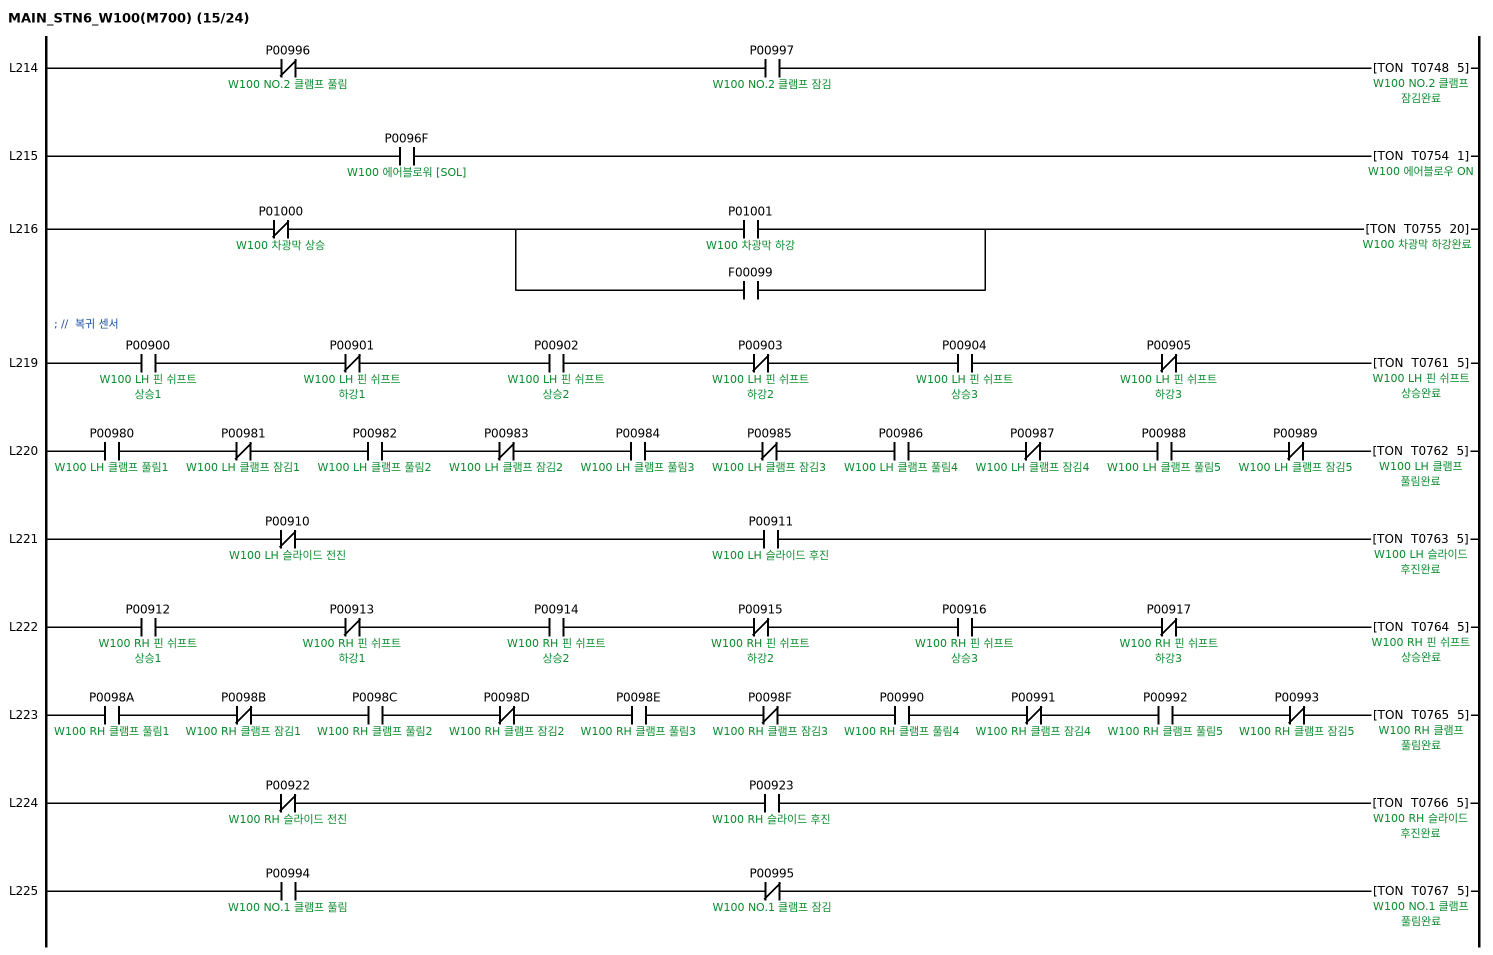
; L214
LOAD NOT  P00996	// W100 NO.2 클램프 풀림
AND       P00997	// W100 NO.2 클램프 잠김
TON       T0748 5	// W100 NO.2 클램프 잠김완료
; L215
LOAD      P0096F	// W100 에어블로워 [SOL]
TON       T0754 1	// W100 에어블로우 ON
; L216
LOAD NOT  P01000	// W100 차광막 상승
LOAD      P01001	// W100 차광막 하강
OR        F00099
AND LOAD
TON       T0755 20	// W100 차광막 하강완료
//   //  복귀 센서
; L219
LOAD      P00900	// W100 LH 핀 쉬프트 상승1
AND NOT   P00901	// W100 LH 핀 쉬프트 하강1
AND       P00902	// W100 LH 핀 쉬프트 상승2
AND NOT   P00903	// W100 LH 핀 쉬프트 하강2
AND       P00904	// W100 LH 핀 쉬프트 상승3
AND NOT   P00905	// W100 LH 핀 쉬프트 하강3
TON       T0761 5	// W100 LH 핀 쉬프트 상승완료
; L220
LOAD      P00980	// W100 LH 클램프 풀림1
AND NOT   P00981	// W100 LH 클램프 잠김1
AND       P00982	// W100 LH 클램프 풀림2
AND NOT   P00983	// W100 LH 클램프 잠김2
AND       P00984	// W100 LH 클램프 풀림3
AND NOT   P00985	// W100 LH 클램프 잠김3
AND       P00986	// W100 LH 클램프 풀림4
AND NOT   P00987	// W100 LH 클램프 잠김4
AND       P00988	// W100 LH 클램프 풀림5
AND NOT   P00989	// W100 LH 클램프 잠김5
TON       T0762 5	// W100 LH 클램프 풀림완료
; L221
LOAD NOT  P00910	// W100 LH 슬라이드 전진
AND       P00911	// W100 LH 슬라이드 후진
TON       T0763 5	// W100 LH 슬라이드 후진완료
; L222
LOAD      P00912	// W100 RH 핀 쉬프트 상승1
AND NOT   P00913	// W100 RH 핀 쉬프트 하강1
AND       P00914	// W100 RH 핀 쉬프트 상승2
AND NOT   P00915	// W100 RH 핀 쉬프트 하강2
AND       P00916	// W100 RH 핀 쉬프트 상승3
AND NOT   P00917	// W100 RH 핀 쉬프트 하강3
TON       T0764 5	// W100 RH 핀 쉬프트 상승완료
; L223
LOAD      P0098A	// W100 RH 클램프 풀림1
AND NOT   P0098B	// W100 RH 클램프 잠김1
AND       P0098C	// W100 RH 클램프 풀림2
AND NOT   P0098D	// W100 RH 클램프 잠김2
AND       P0098E	// W100 RH 클램프 풀림3
AND NOT   P0098F	// W100 RH 클램프 잠김3
AND       P00990	// W100 RH 클램프 풀림4
AND NOT   P00991	// W100 RH 클램프 잠김4
AND       P00992	// W100 RH 클램프 풀림5
AND NOT   P00993	// W100 RH 클램프 잠김5
TON       T0765 5	// W100 RH 클램프 풀림완료
; L224
LOAD NOT  P00922	// W100 RH 슬라이드 전진
AND       P00923	// W100 RH 슬라이드 후진
TON       T0766 5	// W100 RH 슬라이드 후진완료
; L225
LOAD      P00994	// W100 NO.1 클램프 풀림
AND NOT   P00995	// W100 NO.1 클램프 잠김
TON       T0767 5	// W100 NO.1 클램프 풀림완료

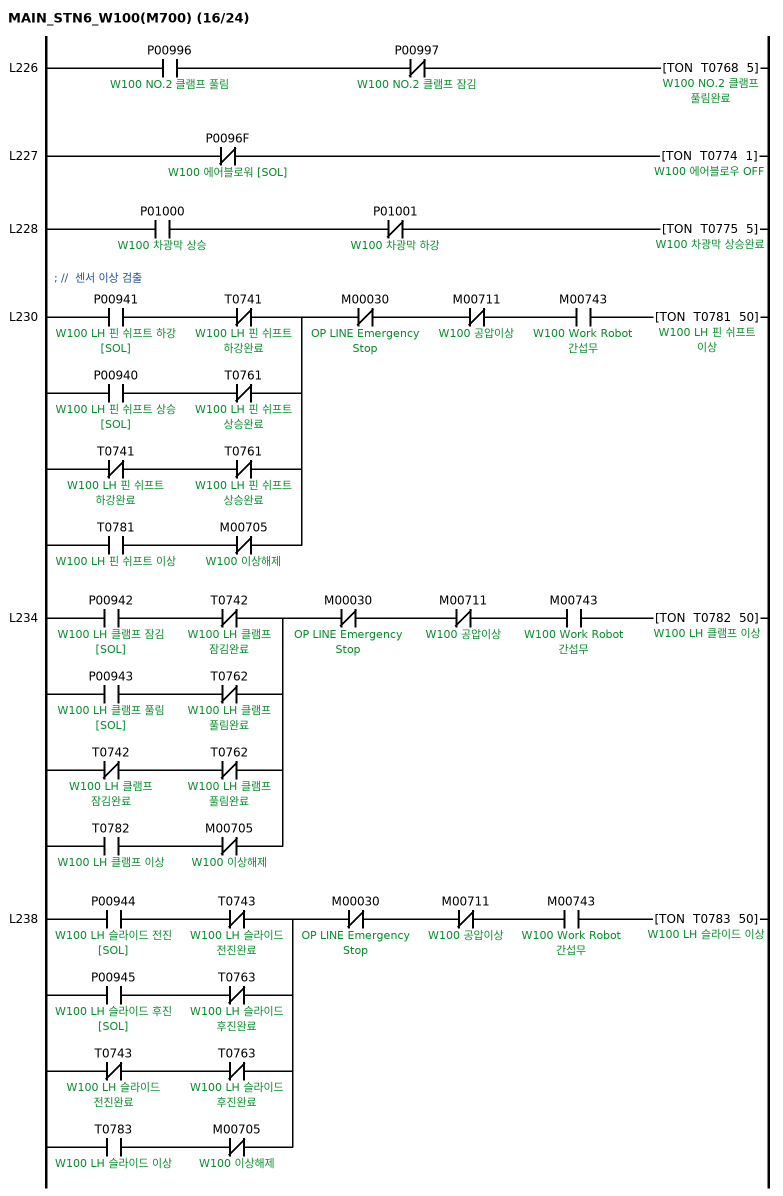
; L226
LOAD      P00996	// W100 NO.2 클램프 풀림
AND NOT   P00997	// W100 NO.2 클램프 잠김
TON       T0768 5	// W100 NO.2 클램프 풀림완료
; L227
LOAD NOT  P0096F	// W100 에어블로워 [SOL]
TON       T0774 1	// W100 에어블로우 OFF
; L228
LOAD      P01000	// W100 차광막 상승
AND NOT   P01001	// W100 차광막 하강
TON       T0775 5	// W100 차광막 상승완료
//     //  센서 이상 검출
; L230
LOAD      P00941	// W100 LH 핀 쉬프트 하강 [SOL]
AND NOT   T0741	// W100 LH 핀 쉬프트 하강완료
LOAD      P00940	// W100 LH 핀 쉬프트 상승 [SOL]
AND NOT   T0761	// W100 LH 핀 쉬프트 상승완료
OR LOAD
LOAD NOT  T0741	// W100 LH 핀 쉬프트 하강완료
AND NOT   T0761	// W100 LH 핀 쉬프트 상승완료
OR LOAD
LOAD      T0781	// W100 LH 핀 쉬프트 이상
AND NOT   M00705	// W100 이상해제
OR LOAD
AND NOT   M00030	// OP LINE Emergency Stop
AND NOT   M00711	// W100 공압이상
AND       M00743	// W100 Work Robot 간섭무
TON       T0781 50	// W100 LH 핀 쉬프트 이상
; L234
LOAD      P00942	// W100 LH 클램프 잠김 [SOL]
AND NOT   T0742	// W100 LH 클램프 잠김완료
LOAD      P00943	// W100 LH 클램프 풀림 [SOL]
AND NOT   T0762	// W100 LH 클램프 풀림완료
OR LOAD
LOAD NOT  T0742	// W100 LH 클램프 잠김완료
AND NOT   T0762	// W100 LH 클램프 풀림완료
OR LOAD
LOAD      T0782	// W100 LH 클램프 이상
AND NOT   M00705	// W100 이상해제
OR LOAD
AND NOT   M00030	// OP LINE Emergency Stop
AND NOT   M00711	// W100 공압이상
AND       M00743	// W100 Work Robot 간섭무
TON       T0782 50	// W100 LH 클램프 이상
; L238
LOAD      P00944	// W100 LH 슬라이드 전진 [SOL]
AND NOT   T0743	// W100 LH 슬라이드 전진완료
LOAD      P00945	// W100 LH 슬라이드 후진 [SOL]
AND NOT   T0763	// W100 LH 슬라이드 후진완료
OR LOAD
LOAD NOT  T0743	// W100 LH 슬라이드 전진완료
AND NOT   T0763	// W100 LH 슬라이드 후진완료
OR LOAD
LOAD      T0783	// W100 LH 슬라이드 이상
AND NOT   M00705	// W100 이상해제
OR LOAD
AND NOT   M00030	// OP LINE Emergency Stop
AND NOT   M00711	// W100 공압이상
AND       M00743	// W100 Work Robot 간섭무
TON       T0783 50	// W100 LH 슬라이드 이상

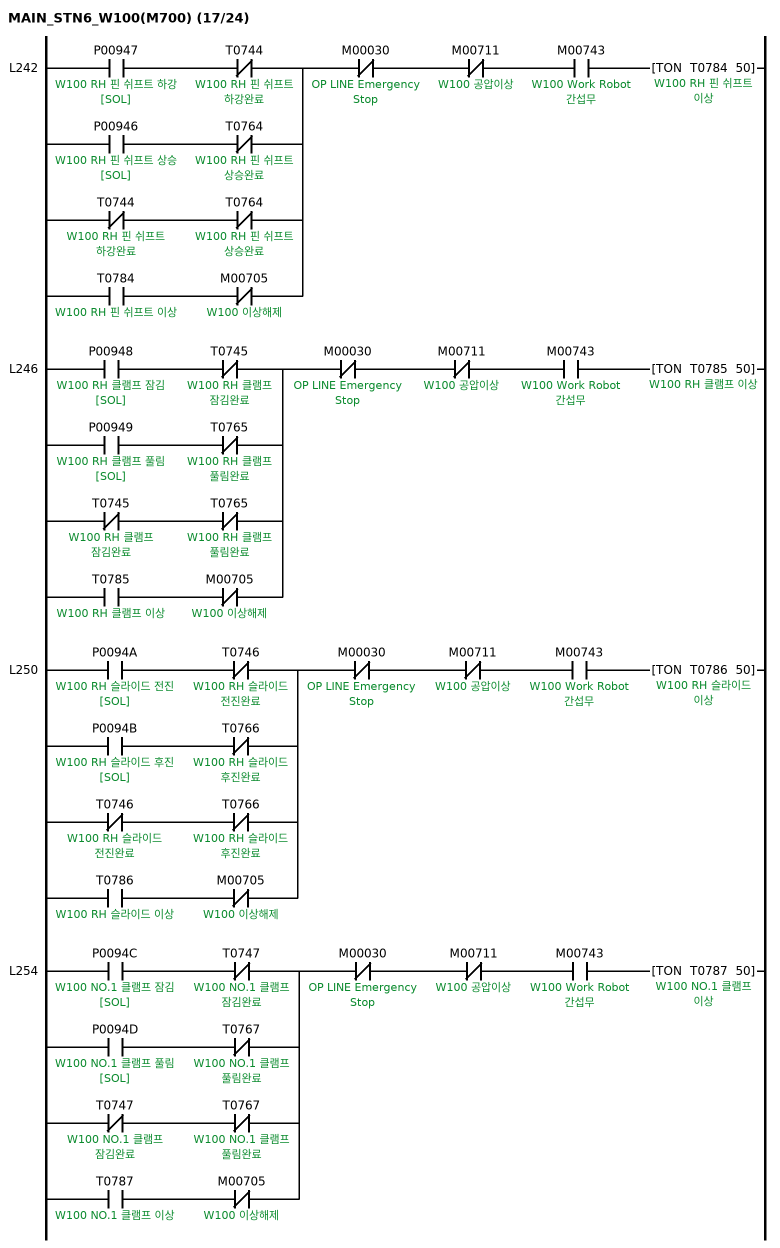
; L242
LOAD      P00947	// W100 RH 핀 쉬프트 하강 [SOL]
AND NOT   T0744	// W100 RH 핀 쉬프트 하강완료
LOAD      P00946	// W100 RH 핀 쉬프트 상승 [SOL]
AND NOT   T0764	// W100 RH 핀 쉬프트 상승완료
OR LOAD
LOAD NOT  T0744	// W100 RH 핀 쉬프트 하강완료
AND NOT   T0764	// W100 RH 핀 쉬프트 상승완료
OR LOAD
LOAD      T0784	// W100 RH 핀 쉬프트 이상
AND NOT   M00705	// W100 이상해제
OR LOAD
AND NOT   M00030	// OP LINE Emergency Stop
AND NOT   M00711	// W100 공압이상
AND       M00743	// W100 Work Robot 간섭무
TON       T0784 50	// W100 RH 핀 쉬프트 이상
; L246
LOAD      P00948	// W100 RH 클램프 잠김 [SOL]
AND NOT   T0745	// W100 RH 클램프 잠김완료
LOAD      P00949	// W100 RH 클램프 풀림 [SOL]
AND NOT   T0765	// W100 RH 클램프 풀림완료
OR LOAD
LOAD NOT  T0745	// W100 RH 클램프 잠김완료
AND NOT   T0765	// W100 RH 클램프 풀림완료
OR LOAD
LOAD      T0785	// W100 RH 클램프 이상
AND NOT   M00705	// W100 이상해제
OR LOAD
AND NOT   M00030	// OP LINE Emergency Stop
AND NOT   M00711	// W100 공압이상
AND       M00743	// W100 Work Robot 간섭무
TON       T0785 50	// W100 RH 클램프 이상
; L250
LOAD      P0094A	// W100 RH 슬라이드 전진 [SOL]
AND NOT   T0746	// W100 RH 슬라이드 전진완료
LOAD      P0094B	// W100 RH 슬라이드 후진 [SOL]
AND NOT   T0766	// W100 RH 슬라이드 후진완료
OR LOAD
LOAD NOT  T0746	// W100 RH 슬라이드 전진완료
AND NOT   T0766	// W100 RH 슬라이드 후진완료
OR LOAD
LOAD      T0786	// W100 RH 슬라이드 이상
AND NOT   M00705	// W100 이상해제
OR LOAD
AND NOT   M00030	// OP LINE Emergency Stop
AND NOT   M00711	// W100 공압이상
AND       M00743	// W100 Work Robot 간섭무
TON       T0786 50	// W100 RH 슬라이드 이상
; L254
LOAD      P0094C	// W100 NO.1 클램프 잠김 [SOL]
AND NOT   T0747	// W100 NO.1 클램프 잠김완료
LOAD      P0094D	// W100 NO.1 클램프 풀림 [SOL]
AND NOT   T0767	// W100 NO.1 클램프 풀림완료
OR LOAD
LOAD NOT  T0747	// W100 NO.1 클램프 잠김완료
AND NOT   T0767	// W100 NO.1 클램프 풀림완료
OR LOAD
LOAD      T0787	// W100 NO.1 클램프 이상
AND NOT   M00705	// W100 이상해제
OR LOAD
AND NOT   M00030	// OP LINE Emergency Stop
AND NOT   M00711	// W100 공압이상
AND       M00743	// W100 Work Robot 간섭무
TON       T0787 50	// W100 NO.1 클램프 이상

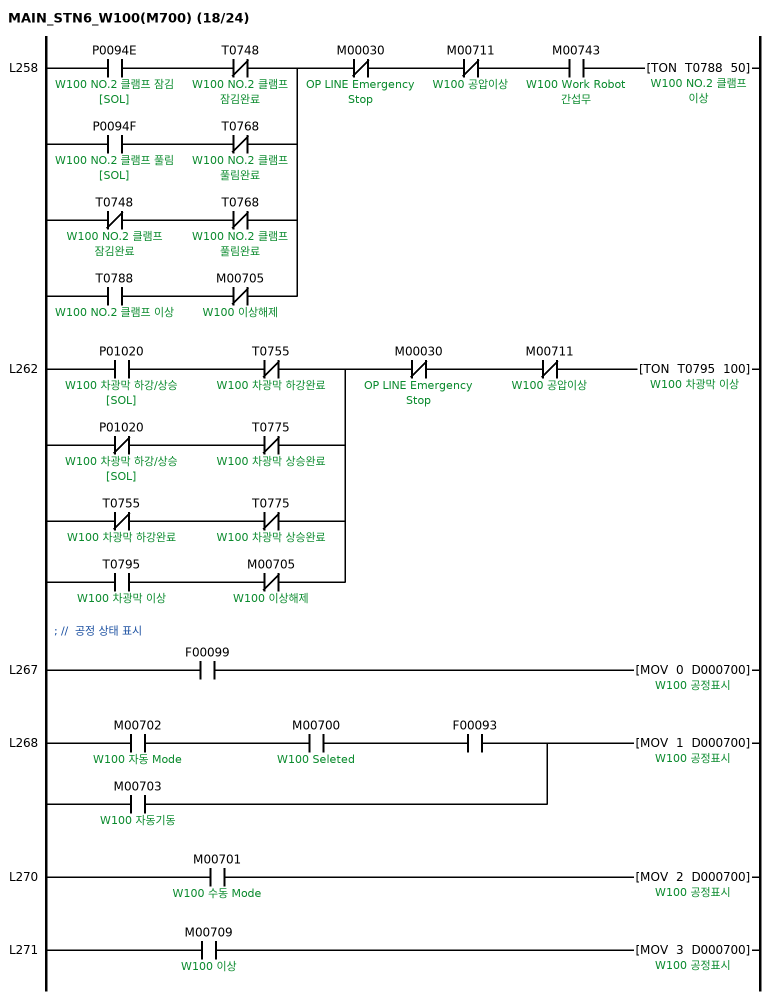
; L258
LOAD      P0094E	// W100 NO.2 클램프 잠김 [SOL]
AND NOT   T0748	// W100 NO.2 클램프 잠김완료
LOAD      P0094F	// W100 NO.2 클램프 풀림 [SOL]
AND NOT   T0768	// W100 NO.2 클램프 풀림완료
OR LOAD
LOAD NOT  T0748	// W100 NO.2 클램프 잠김완료
AND NOT   T0768	// W100 NO.2 클램프 풀림완료
OR LOAD
LOAD      T0788	// W100 NO.2 클램프 이상
AND NOT   M00705	// W100 이상해제
OR LOAD
AND NOT   M00030	// OP LINE Emergency Stop
AND NOT   M00711	// W100 공압이상
AND       M00743	// W100 Work Robot 간섭무
TON       T0788 50	// W100 NO.2 클램프 이상
; L262
LOAD      P01020	// W100 차광막 하강/상승 [SOL]
AND NOT   T0755	// W100 차광막 하강완료
LOAD NOT  P01020	// W100 차광막 하강/상승 [SOL]
AND NOT   T0775	// W100 차광막 상승완료
OR LOAD
LOAD NOT  T0755	// W100 차광막 하강완료
AND NOT   T0775	// W100 차광막 상승완료
OR LOAD
LOAD      T0795	// W100 차광막 이상
AND NOT   M00705	// W100 이상해제
OR LOAD
AND NOT   M00030	// OP LINE Emergency Stop
AND NOT   M00711	// W100 공압이상
TON       T0795 100	// W100 차광막 이상
//   //  공정 상태 표시
; L267
LOAD      F00099
MOV       0 D000700	// W100 공정표시
; L268
LOAD      M00702	// W100 자동 Mode
AND       M00700	// W100 Seleted
AND       F00093
OR        M00703	// W100 자동기동
MOV       1 D000700	// W100 공정표시
; L270
LOAD      M00701	// W100 수동 Mode
MOV       2 D000700	// W100 공정표시
; L271
LOAD      M00709	// W100 이상
MOV       3 D000700	// W100 공정표시

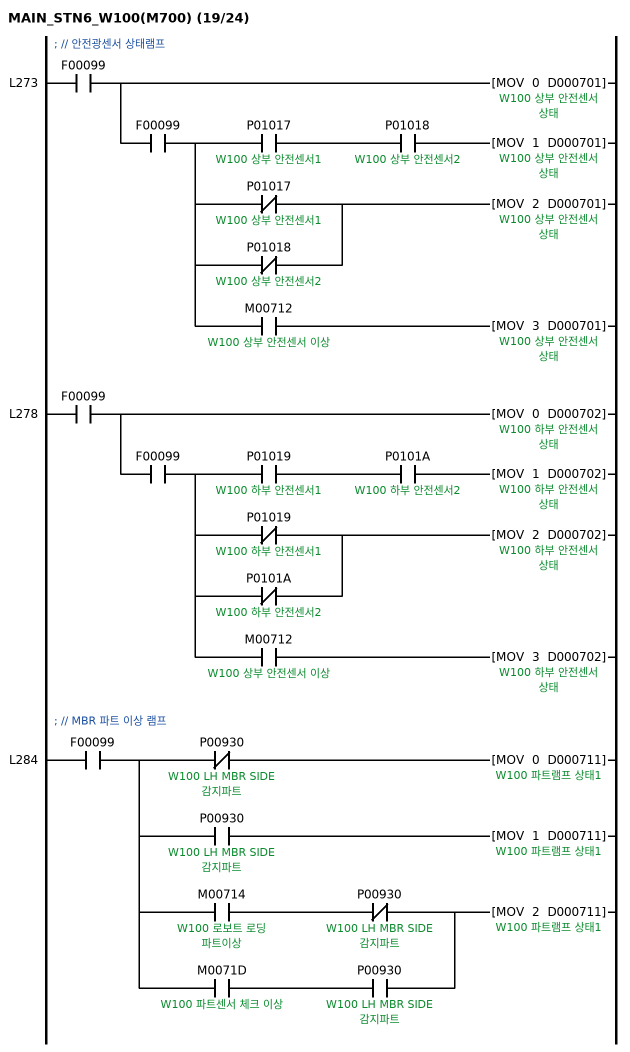
//   // 안전광센서 상태램프
; L273
LOAD      F00099
MOV       0 D000701	// W100 상부 안전센서 상태
AND       F00099
MPUSH
AND       P01017	// W100 상부 안전센서1
AND       P01018	// W100 상부 안전센서2
MOV       1 D000701	// W100 상부 안전센서 상태
MLOAD
LOAD NOT  P01017	// W100 상부 안전센서1
OR NOT    P01018	// W100 상부 안전센서2
AND LOAD
MOV       2 D000701	// W100 상부 안전센서 상태
MPOP
AND       M00712	// W100 상부 안전센서 이상
MOV       3 D000701	// W100 상부 안전센서 상태
; L278
LOAD      F00099
MOV       0 D000702	// W100 하부 안전센서 상태
AND       F00099
MPUSH
AND       P01019	// W100 하부 안전센서1
AND       P0101A	// W100 하부 안전센서2
MOV       1 D000702	// W100 하부 안전센서 상태
MLOAD
LOAD NOT  P01019	// W100 하부 안전센서1
OR NOT    P0101A	// W100 하부 안전센서2
AND LOAD
MOV       2 D000702	// W100 하부 안전센서 상태
MPOP
AND       M00712	// W100 상부 안전센서 이상
MOV       3 D000702	// W100 하부 안전센서 상태
//   // MBR 파트 이상 램프
; L284
LOAD      F00099
MPUSH
AND NOT   P00930	// W100 LH MBR SIDE 감지파트
MOV       0 D000711	// W100 파트램프 상태1
MLOAD
AND       P00930	// W100 LH MBR SIDE 감지파트
MOV       1 D000711	// W100 파트램프 상태1
MPOP
LOAD      M00714	// W100 로보트 로딩 파트이상
AND NOT   P00930	// W100 LH MBR SIDE 감지파트
LOAD      M0071D	// W100 파트센서 체크 이상
AND       P00930	// W100 LH MBR SIDE 감지파트
OR LOAD
AND LOAD
MOV       2 D000711	// W100 파트램프 상태1

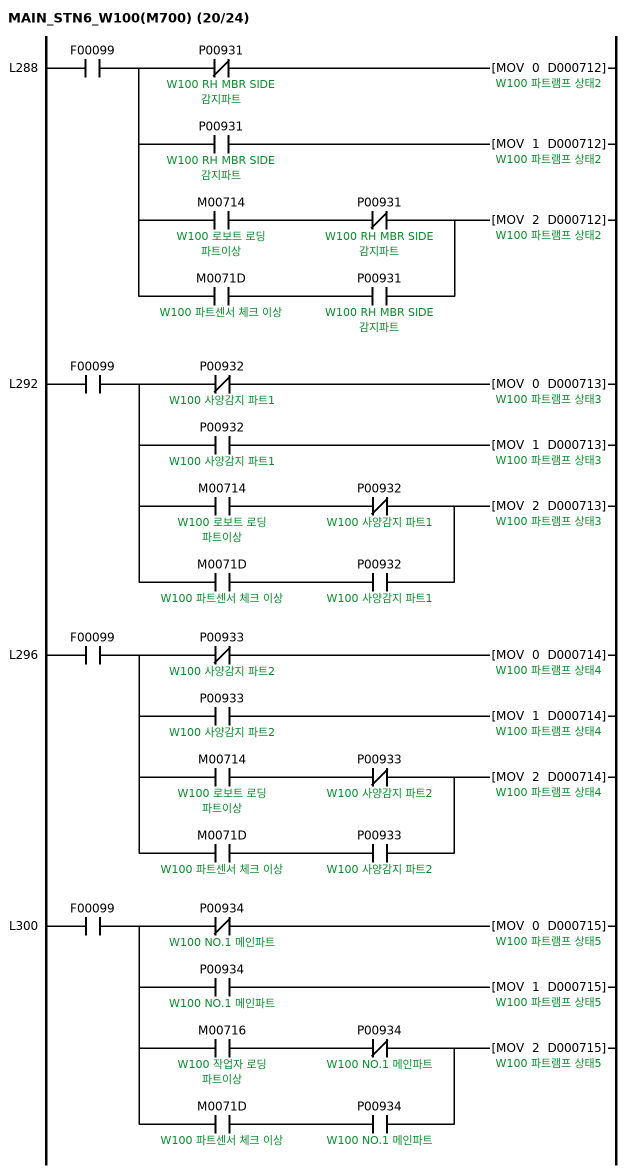
; L288
LOAD      F00099
MPUSH
AND NOT   P00931	// W100 RH MBR SIDE 감지파트
MOV       0 D000712	// W100 파트램프 상태2
MLOAD
AND       P00931	// W100 RH MBR SIDE 감지파트
MOV       1 D000712	// W100 파트램프 상태2
MPOP
LOAD      M00714	// W100 로보트 로딩 파트이상
AND NOT   P00931	// W100 RH MBR SIDE 감지파트
LOAD      M0071D	// W100 파트센서 체크 이상
AND       P00931	// W100 RH MBR SIDE 감지파트
OR LOAD
AND LOAD
MOV       2 D000712	// W100 파트램프 상태2
; L292
LOAD      F00099
MPUSH
AND NOT   P00932	// W100 사양감지 파트1
MOV       0 D000713	// W100 파트램프 상태3
MLOAD
AND       P00932	// W100 사양감지 파트1
MOV       1 D000713	// W100 파트램프 상태3
MPOP
LOAD      M00714	// W100 로보트 로딩 파트이상
AND NOT   P00932	// W100 사양감지 파트1
LOAD      M0071D	// W100 파트센서 체크 이상
AND       P00932	// W100 사양감지 파트1
OR LOAD
AND LOAD
MOV       2 D000713	// W100 파트램프 상태3
; L296
LOAD      F00099
MPUSH
AND NOT   P00933	// W100 사양감지 파트2
MOV       0 D000714	// W100 파트램프 상태4
MLOAD
AND       P00933	// W100 사양감지 파트2
MOV       1 D000714	// W100 파트램프 상태4
MPOP
LOAD      M00714	// W100 로보트 로딩 파트이상
AND NOT   P00933	// W100 사양감지 파트2
LOAD      M0071D	// W100 파트센서 체크 이상
AND       P00933	// W100 사양감지 파트2
OR LOAD
AND LOAD
MOV       2 D000714	// W100 파트램프 상태4
; L300
LOAD      F00099
MPUSH
AND NOT   P00934	// W100 NO.1 메인파트
MOV       0 D000715	// W100 파트램프 상태5
MLOAD
AND       P00934	// W100 NO.1 메인파트
MOV       1 D000715	// W100 파트램프 상태5
MPOP
LOAD      M00716	// W100 작업자 로딩 파트이상
AND NOT   P00934	// W100 NO.1 메인파트
LOAD      M0071D	// W100 파트센서 체크 이상
AND       P00934	// W100 NO.1 메인파트
OR LOAD
AND LOAD
MOV       2 D000715	// W100 파트램프 상태5

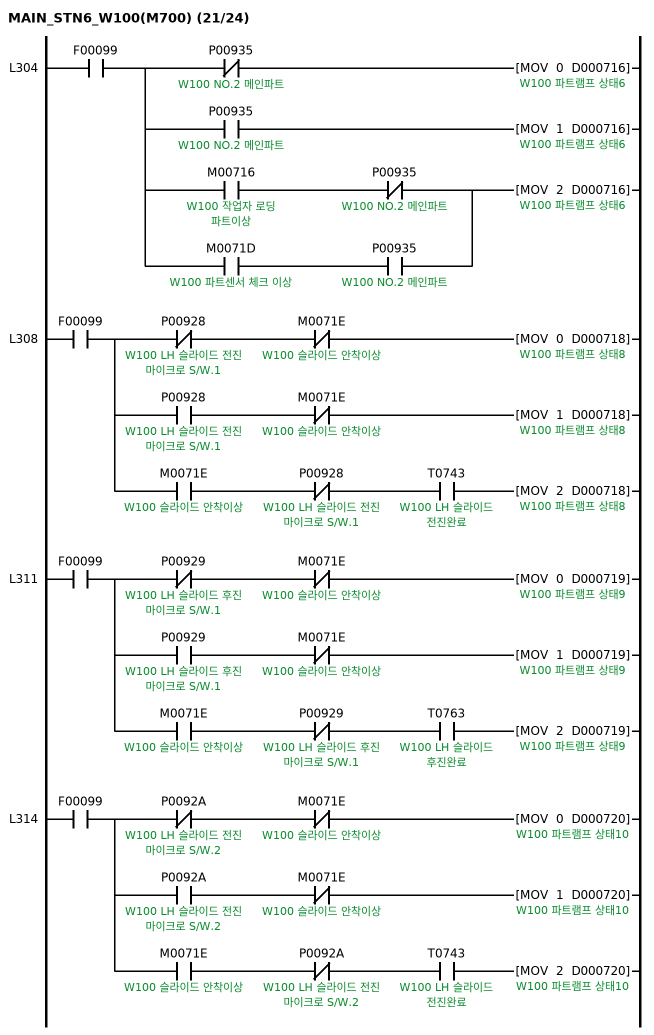
; L304
LOAD      F00099
MPUSH
AND NOT   P00935	// W100 NO.2 메인파트
MOV       0 D000716	// W100 파트램프 상태6
MLOAD
AND       P00935	// W100 NO.2 메인파트
MOV       1 D000716	// W100 파트램프 상태6
MPOP
LOAD      M00716	// W100 작업자 로딩 파트이상
AND NOT   P00935	// W100 NO.2 메인파트
LOAD      M0071D	// W100 파트센서 체크 이상
AND       P00935	// W100 NO.2 메인파트
OR LOAD
AND LOAD
MOV       2 D000716	// W100 파트램프 상태6
; L308
LOAD      F00099
MPUSH
AND NOT   P00928	// W100 LH 슬라이드 전진 마이크로 S/W.1
AND NOT   M0071E	// W100 슬라이드 안착이상
MOV       0 D000718	// W100 파트램프 상태8
MLOAD
AND       P00928	// W100 LH 슬라이드 전진 마이크로 S/W.1
AND NOT   M0071E	// W100 슬라이드 안착이상
MOV       1 D000718	// W100 파트램프 상태8
MPOP
AND       M0071E	// W100 슬라이드 안착이상
AND NOT   P00928	// W100 LH 슬라이드 전진 마이크로 S/W.1
AND       T0743	// W100 LH 슬라이드 전진완료
MOV       2 D000718	// W100 파트램프 상태8
; L311
LOAD      F00099
MPUSH
AND NOT   P00929	// W100 LH 슬라이드 후진 마이크로 S/W.1
AND NOT   M0071E	// W100 슬라이드 안착이상
MOV       0 D000719	// W100 파트램프 상태9
MLOAD
AND       P00929	// W100 LH 슬라이드 후진 마이크로 S/W.1
AND NOT   M0071E	// W100 슬라이드 안착이상
MOV       1 D000719	// W100 파트램프 상태9
MPOP
AND       M0071E	// W100 슬라이드 안착이상
AND NOT   P00929	// W100 LH 슬라이드 후진 마이크로 S/W.1
AND       T0763	// W100 LH 슬라이드 후진완료
MOV       2 D000719	// W100 파트램프 상태9
; L314
LOAD      F00099
MPUSH
AND NOT   P0092A	// W100 LH 슬라이드 전진 마이크로 S/W.2
AND NOT   M0071E	// W100 슬라이드 안착이상
MOV       0 D000720	// W100 파트램프 상태10
MLOAD
AND       P0092A	// W100 LH 슬라이드 전진 마이크로 S/W.2
AND NOT   M0071E	// W100 슬라이드 안착이상
MOV       1 D000720	// W100 파트램프 상태10
MPOP
AND       M0071E	// W100 슬라이드 안착이상
AND NOT   P0092A	// W100 LH 슬라이드 전진 마이크로 S/W.2
AND       T0743	// W100 LH 슬라이드 전진완료
MOV       2 D000720	// W100 파트램프 상태10

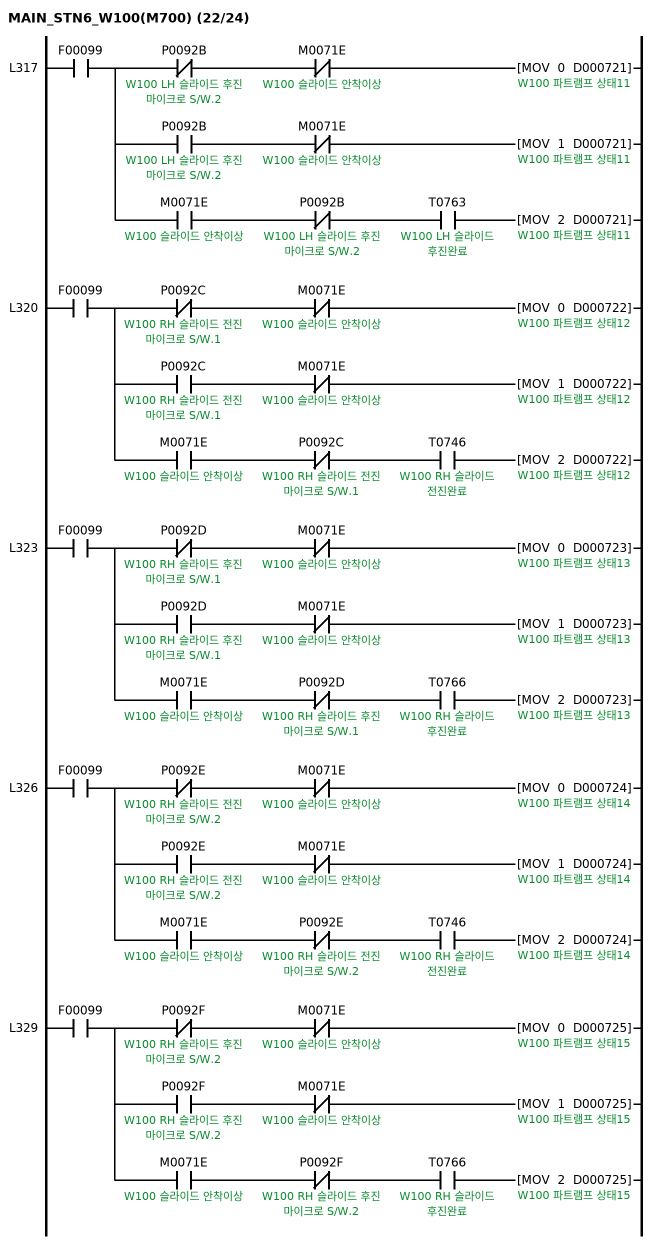
; L317
LOAD      F00099
MPUSH
AND NOT   P0092B	// W100 LH 슬라이드 후진 마이크로 S/W.2
AND NOT   M0071E	// W100 슬라이드 안착이상
MOV       0 D000721	// W100 파트램프 상태11
MLOAD
AND       P0092B	// W100 LH 슬라이드 후진 마이크로 S/W.2
AND NOT   M0071E	// W100 슬라이드 안착이상
MOV       1 D000721	// W100 파트램프 상태11
MPOP
AND       M0071E	// W100 슬라이드 안착이상
AND NOT   P0092B	// W100 LH 슬라이드 후진 마이크로 S/W.2
AND       T0763	// W100 LH 슬라이드 후진완료
MOV       2 D000721	// W100 파트램프 상태11
; L320
LOAD      F00099
MPUSH
AND NOT   P0092C	// W100 RH 슬라이드 전진 마이크로 S/W.1
AND NOT   M0071E	// W100 슬라이드 안착이상
MOV       0 D000722	// W100 파트램프 상태12
MLOAD
AND       P0092C	// W100 RH 슬라이드 전진 마이크로 S/W.1
AND NOT   M0071E	// W100 슬라이드 안착이상
MOV       1 D000722	// W100 파트램프 상태12
MPOP
AND       M0071E	// W100 슬라이드 안착이상
AND NOT   P0092C	// W100 RH 슬라이드 전진 마이크로 S/W.1
AND       T0746	// W100 RH 슬라이드 전진완료
MOV       2 D000722	// W100 파트램프 상태12
; L323
LOAD      F00099
MPUSH
AND NOT   P0092D	// W100 RH 슬라이드 후진 마이크로 S/W.1
AND NOT   M0071E	// W100 슬라이드 안착이상
MOV       0 D000723	// W100 파트램프 상태13
MLOAD
AND       P0092D	// W100 RH 슬라이드 후진 마이크로 S/W.1
AND NOT   M0071E	// W100 슬라이드 안착이상
MOV       1 D000723	// W100 파트램프 상태13
MPOP
AND       M0071E	// W100 슬라이드 안착이상
AND NOT   P0092D	// W100 RH 슬라이드 후진 마이크로 S/W.1
AND       T0766	// W100 RH 슬라이드 후진완료
MOV       2 D000723	// W100 파트램프 상태13
; L326
LOAD      F00099
MPUSH
AND NOT   P0092E	// W100 RH 슬라이드 전진 마이크로 S/W.2
AND NOT   M0071E	// W100 슬라이드 안착이상
MOV       0 D000724	// W100 파트램프 상태14
MLOAD
AND       P0092E	// W100 RH 슬라이드 전진 마이크로 S/W.2
AND NOT   M0071E	// W100 슬라이드 안착이상
MOV       1 D000724	// W100 파트램프 상태14
MPOP
AND       M0071E	// W100 슬라이드 안착이상
AND NOT   P0092E	// W100 RH 슬라이드 전진 마이크로 S/W.2
AND       T0746	// W100 RH 슬라이드 전진완료
MOV       2 D000724	// W100 파트램프 상태14
; L329
LOAD      F00099
MPUSH
AND NOT   P0092F	// W100 RH 슬라이드 후진 마이크로 S/W.2
AND NOT   M0071E	// W100 슬라이드 안착이상
MOV       0 D000725	// W100 파트램프 상태15
MLOAD
AND       P0092F	// W100 RH 슬라이드 후진 마이크로 S/W.2
AND NOT   M0071E	// W100 슬라이드 안착이상
MOV       1 D000725	// W100 파트램프 상태15
MPOP
AND       M0071E	// W100 슬라이드 안착이상
AND NOT   P0092F	// W100 RH 슬라이드 후진 마이크로 S/W.2
AND       T0766	// W100 RH 슬라이드 후진완료
MOV       2 D000725	// W100 파트램프 상태15

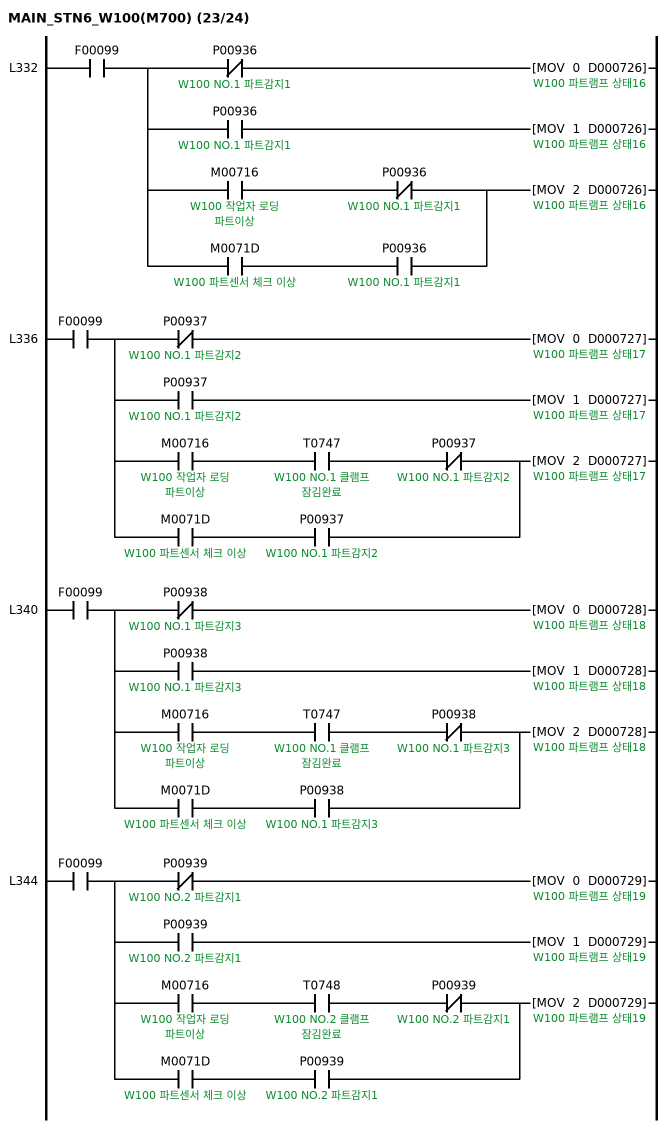
; L332
LOAD      F00099
MPUSH
AND NOT   P00936	// W100 NO.1 파트감지1
MOV       0 D000726	// W100 파트램프 상태16
MLOAD
AND       P00936	// W100 NO.1 파트감지1
MOV       1 D000726	// W100 파트램프 상태16
MPOP
LOAD      M00716	// W100 작업자 로딩 파트이상
AND NOT   P00936	// W100 NO.1 파트감지1
LOAD      M0071D	// W100 파트센서 체크 이상
AND       P00936	// W100 NO.1 파트감지1
OR LOAD
AND LOAD
MOV       2 D000726	// W100 파트램프 상태16
; L336
LOAD      F00099
MPUSH
AND NOT   P00937	// W100 NO.1 파트감지2
MOV       0 D000727	// W100 파트램프 상태17
MLOAD
AND       P00937	// W100 NO.1 파트감지2
MOV       1 D000727	// W100 파트램프 상태17
MPOP
LOAD      M00716	// W100 작업자 로딩 파트이상
AND       T0747	// W100 NO.1 클램프 잠김완료
AND NOT   P00937	// W100 NO.1 파트감지2
LOAD      M0071D	// W100 파트센서 체크 이상
AND       P00937	// W100 NO.1 파트감지2
OR LOAD
AND LOAD
MOV       2 D000727	// W100 파트램프 상태17
; L340
LOAD      F00099
MPUSH
AND NOT   P00938	// W100 NO.1 파트감지3
MOV       0 D000728	// W100 파트램프 상태18
MLOAD
AND       P00938	// W100 NO.1 파트감지3
MOV       1 D000728	// W100 파트램프 상태18
MPOP
LOAD      M00716	// W100 작업자 로딩 파트이상
AND       T0747	// W100 NO.1 클램프 잠김완료
AND NOT   P00938	// W100 NO.1 파트감지3
LOAD      M0071D	// W100 파트센서 체크 이상
AND       P00938	// W100 NO.1 파트감지3
OR LOAD
AND LOAD
MOV       2 D000728	// W100 파트램프 상태18
; L344
LOAD      F00099
MPUSH
AND NOT   P00939	// W100 NO.2 파트감지1
MOV       0 D000729	// W100 파트램프 상태19
MLOAD
AND       P00939	// W100 NO.2 파트감지1
MOV       1 D000729	// W100 파트램프 상태19
MPOP
LOAD      M00716	// W100 작업자 로딩 파트이상
AND       T0748	// W100 NO.2 클램프 잠김완료
AND NOT   P00939	// W100 NO.2 파트감지1
LOAD      M0071D	// W100 파트센서 체크 이상
AND       P00939	// W100 NO.2 파트감지1
OR LOAD
AND LOAD
MOV       2 D000729	// W100 파트램프 상태19

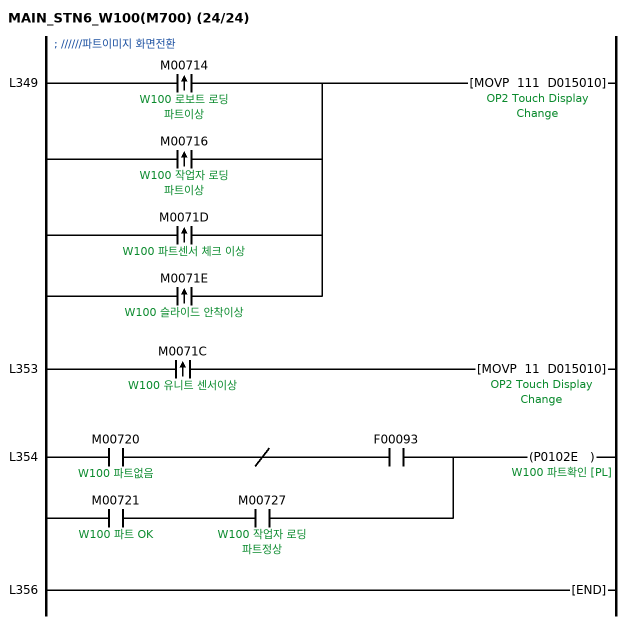
// //////파트이미지 화면전환
; L349
LOADP     M00714	// W100 로보트 로딩 파트이상
ORP       M00716	// W100 작업자 로딩 파트이상
ORP       M0071D	// W100 파트센서 체크 이상
ORP       M0071E	// W100 슬라이드 안착이상
MOVP      111 D015010	// OP2 Touch Display Change
; L353
LOADP     M0071C	// W100 유니트 센서이상
MOVP      11 D015010	// OP2 Touch Display Change
; L354
LOAD      M00720	// W100 파트없음
NOT
AND       F00093
LOAD      M00721	// W100 파트 OK
AND       M00727	// W100 작업자 로딩 파트정상
OR LOAD
OUT       P0102E	// W100 파트확인 [PL]
; L356
END

PROGRAM MAIN_STN7_W130(M1400) (task: 스캔 프로그램)

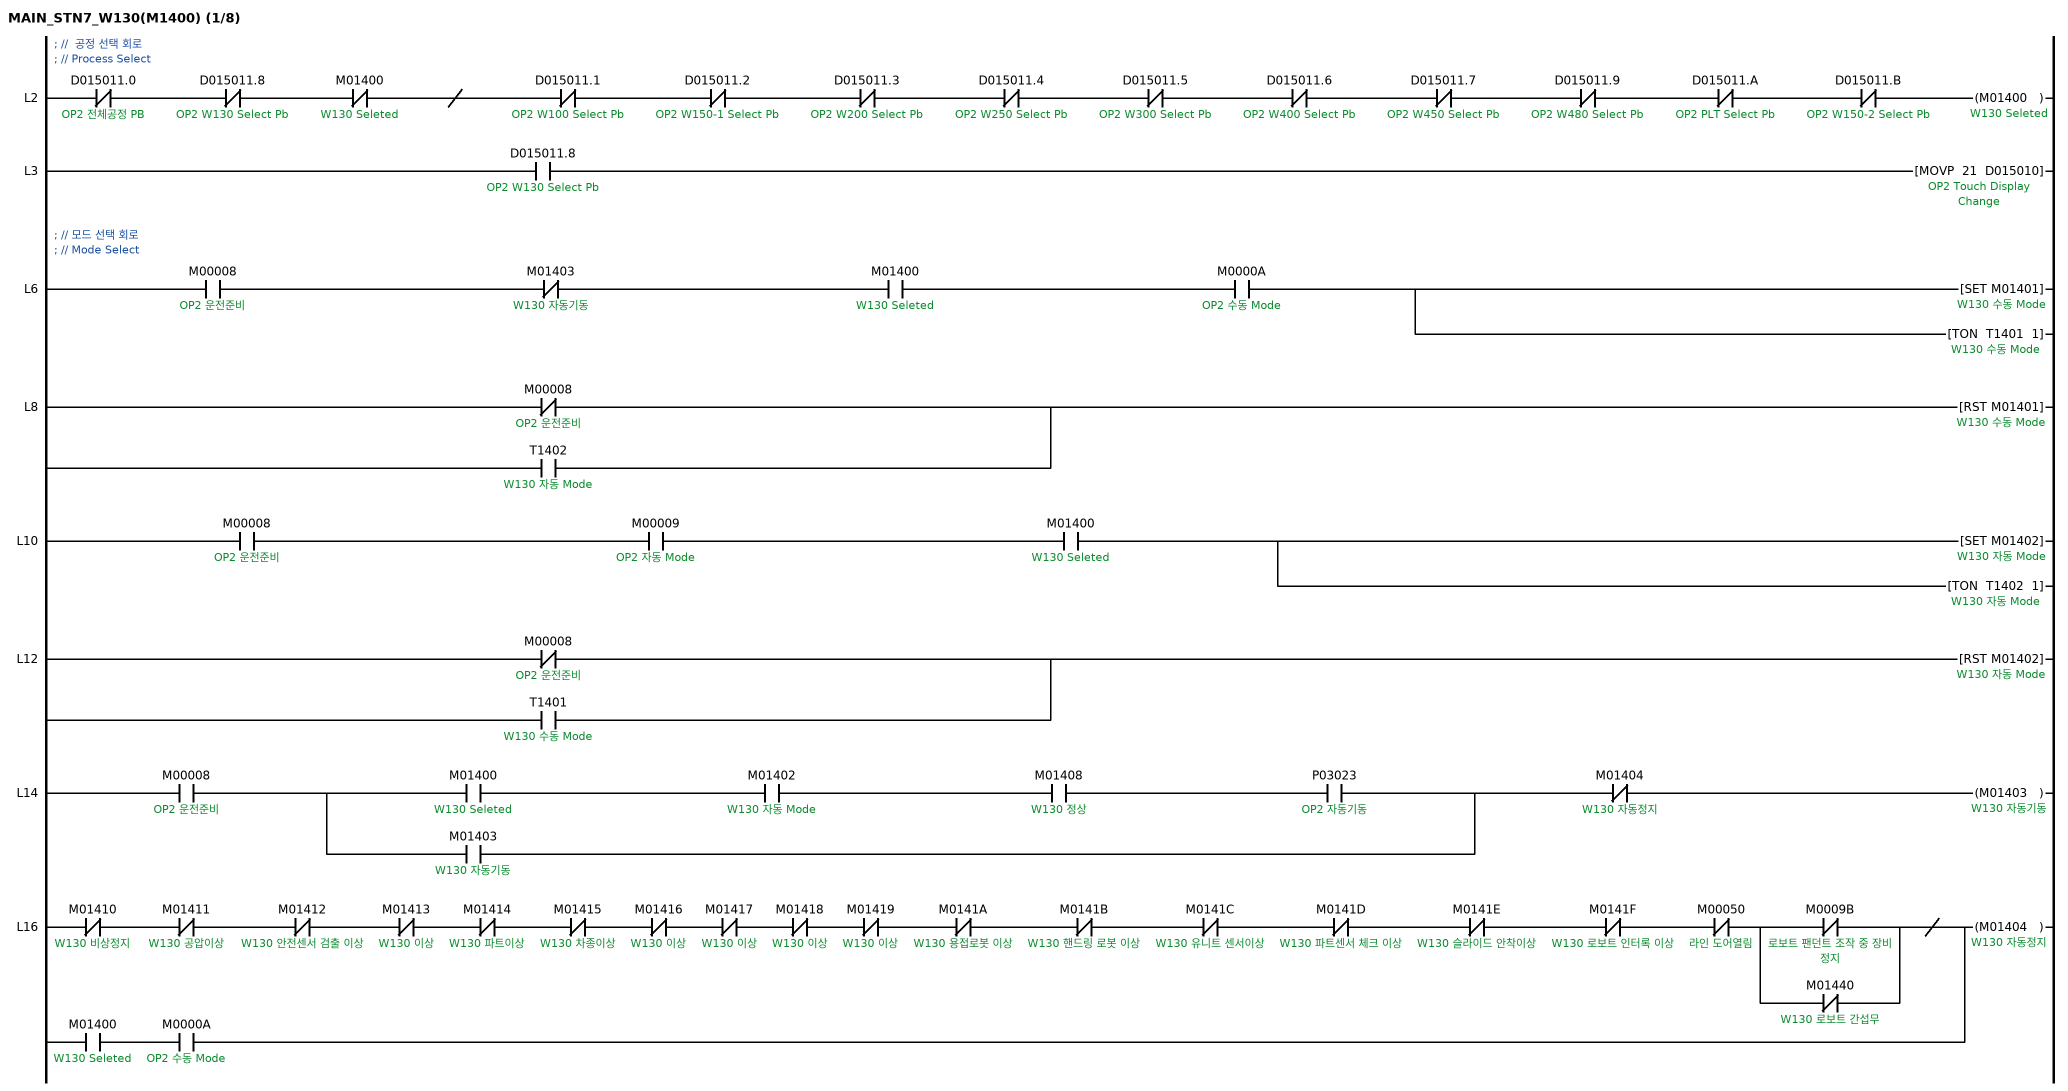
//   //  공정 선택 회로
//   // Process Select
; L2
LOAD NOT  D015011.0	// OP2 전체공정 PB
AND NOT   D015011.8	// OP2 W130 Select Pb
AND NOT   M01400	// W130 Seleted
NOT
AND NOT   D015011.1	// OP2 W100 Select Pb
AND NOT   D015011.2	// OP2 W150-1 Select Pb
AND NOT   D015011.3	// OP2 W200 Select Pb
AND NOT   D015011.4	// OP2 W250 Select Pb
AND NOT   D015011.5	// OP2 W300 Select Pb
AND NOT   D015011.6	// OP2 W400 Select Pb
AND NOT   D015011.7	// OP2 W450 Select Pb
AND NOT   D015011.9	// OP2 W480 Select Pb
AND NOT   D015011.A	// OP2 PLT Select Pb
AND NOT   D015011.B	// OP2 W150-2 Select Pb
OUT       M01400	// W130 Seleted
; L3
LOAD      D015011.8	// OP2 W130 Select Pb
MOVP      21 D015010	// OP2 Touch Display Change
// // 모드 선택 회로
//   // Mode Select
; L6
LOAD      M00008	// OP2 운전준비
AND NOT   M01403	// W130 자동기동
AND       M01400	// W130 Seleted
AND       M0000A	// OP2 수동 Mode
SET       M01401	// W130 수동 Mode
TON       T1401 1	// W130 수동 Mode
; L8
LOAD NOT  M00008	// OP2 운전준비
OR        T1402	// W130 자동 Mode
RST       M01401	// W130 수동 Mode
; L10
LOAD      M00008	// OP2 운전준비
AND       M00009	// OP2 자동 Mode
AND       M01400	// W130 Seleted
SET       M01402	// W130 자동 Mode
TON       T1402 1	// W130 자동 Mode
; L12
LOAD NOT  M00008	// OP2 운전준비
OR        T1401	// W130 수동 Mode
RST       M01402	// W130 자동 Mode
; L14
LOAD      M00008	// OP2 운전준비
LOAD      M01400	// W130 Seleted
AND       M01402	// W130 자동 Mode
AND       M01408	// W130 정상
AND       P03023	// OP2 자동기동
OR        M01403	// W130 자동기동
AND LOAD
AND NOT   M01404	// W130 자동정지
OUT       M01403	// W130 자동기동
; L16
LOAD NOT  M01410	// W130 비상정지
AND NOT   M01411	// W130 공압이상
AND NOT   M01412	// W130 안전센서 검출 이상
AND NOT   M01413	// W130 이상
AND NOT   M01414	// W130 파트이상
AND NOT   M01415	// W130 차종이상
AND NOT   M01416	// W130 이상
AND NOT   M01417	// W130 이상
AND NOT   M01418	// W130 이상
AND NOT   M01419	// W130 이상
AND NOT   M0141A	// W130 용접로봇 이상
AND NOT   M0141B	// W130 핸드링 로봇 이상
AND NOT   M0141C	// W130 유니트 센서이상
AND NOT   M0141D	// W130 파트센서 체크 이상
AND NOT   M0141E	// W130 슬라이드 안착이상
AND NOT   M0141F	// W130 로보트 인터록 이상
AND NOT   M00050	// 라인 도어열림
LOAD NOT  M0009B	// 로보트 팬던트 조작 중 장비 정지
OR NOT    M01440	// W130 로보트 간섭무
AND LOAD
NOT
LOAD      M01400	// W130 Seleted
AND       M0000A	// OP2 수동 Mode
OR LOAD
OUT       M01404	// W130 자동정지

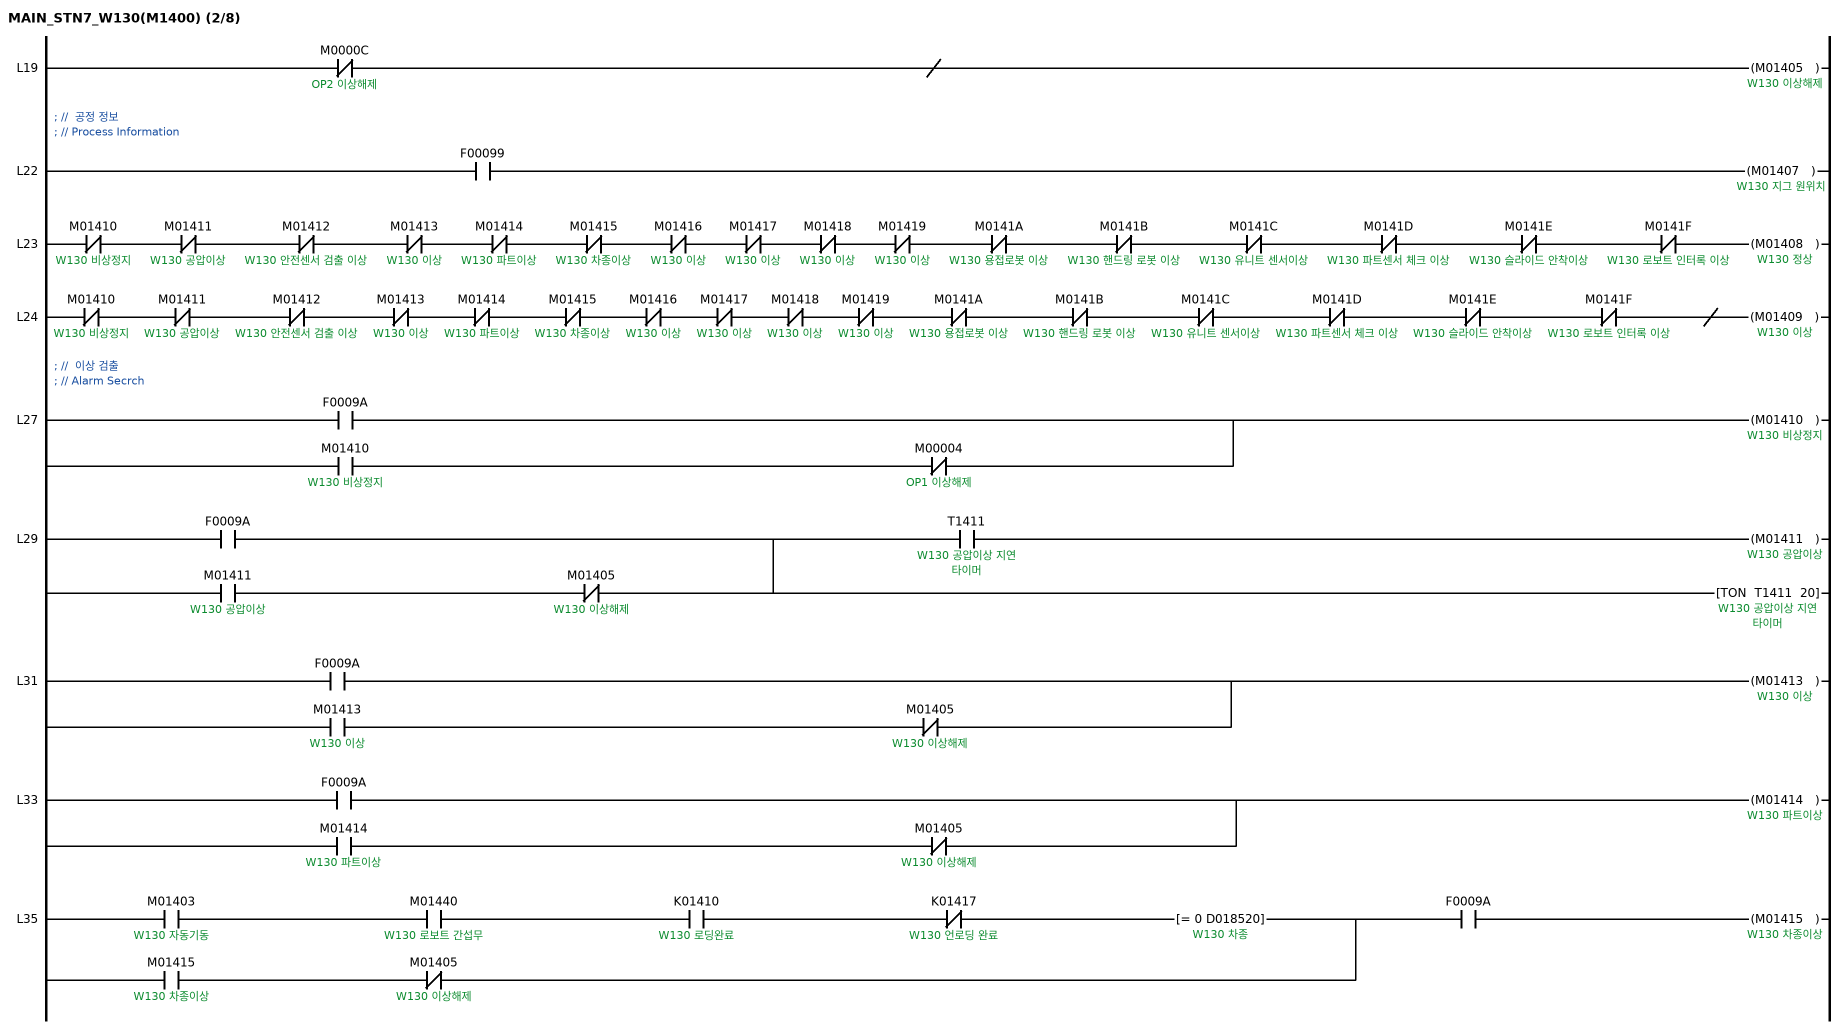
; L19
LOAD NOT  M0000C	// OP2 이상해제
NOT
OUT       M01405	// W130 이상해제
//   //  공정 정보
//   // Process Information
; L22
LOAD      F00099
OUT       M01407	// W130 지그 원위치
; L23
LOAD NOT  M01410	// W130 비상정지
AND NOT   M01411	// W130 공압이상
AND NOT   M01412	// W130 안전센서 검출 이상
AND NOT   M01413	// W130 이상
AND NOT   M01414	// W130 파트이상
AND NOT   M01415	// W130 차종이상
AND NOT   M01416	// W130 이상
AND NOT   M01417	// W130 이상
AND NOT   M01418	// W130 이상
AND NOT   M01419	// W130 이상
AND NOT   M0141A	// W130 용접로봇 이상
AND NOT   M0141B	// W130 핸드링 로봇 이상
AND NOT   M0141C	// W130 유니트 센서이상
AND NOT   M0141D	// W130 파트센서 체크 이상
AND NOT   M0141E	// W130 슬라이드 안착이상
AND NOT   M0141F	// W130 로보트 인터록 이상
OUT       M01408	// W130 정상
; L24
LOAD NOT  M01410	// W130 비상정지
AND NOT   M01411	// W130 공압이상
AND NOT   M01412	// W130 안전센서 검출 이상
AND NOT   M01413	// W130 이상
AND NOT   M01414	// W130 파트이상
AND NOT   M01415	// W130 차종이상
AND NOT   M01416	// W130 이상
AND NOT   M01417	// W130 이상
AND NOT   M01418	// W130 이상
AND NOT   M01419	// W130 이상
AND NOT   M0141A	// W130 용접로봇 이상
AND NOT   M0141B	// W130 핸드링 로봇 이상
AND NOT   M0141C	// W130 유니트 센서이상
AND NOT   M0141D	// W130 파트센서 체크 이상
AND NOT   M0141E	// W130 슬라이드 안착이상
AND NOT   M0141F	// W130 로보트 인터록 이상
NOT
OUT       M01409	// W130 이상
//   //  이상 검출
//   // Alarm Secrch
; L27
LOAD      F0009A
LOAD      M01410	// W130 비상정지
AND NOT   M00004	// OP1 이상해제
OR LOAD
OUT       M01410	// W130 비상정지
; L29
LOAD      F0009A
LOAD      M01411	// W130 공압이상
AND NOT   M01405	// W130 이상해제
OR LOAD
MPUSH
AND       T1411	// W130 공압이상 지연 타이머
OUT       M01411	// W130 공압이상
MPOP
TON       T1411 20	// W130 공압이상 지연 타이머
; L31
LOAD      F0009A
LOAD      M01413	// W130 이상
AND NOT   M01405	// W130 이상해제
OR LOAD
OUT       M01413	// W130 이상
; L33
LOAD      F0009A
LOAD      M01414	// W130 파트이상
AND NOT   M01405	// W130 이상해제
OR LOAD
OUT       M01414	// W130 파트이상
; L35
LOAD      M01403	// W130 자동기동
AND       M01440	// W130 로보트 간섭무
AND       K01410	// W130 로딩완료
AND NOT   K01417	// W130 언로딩 완료
AND=      0 D018520	// W130 차종
LOAD      M01415	// W130 차종이상
AND NOT   M01405	// W130 이상해제
OR LOAD
AND       F0009A
OUT       M01415	// W130 차종이상

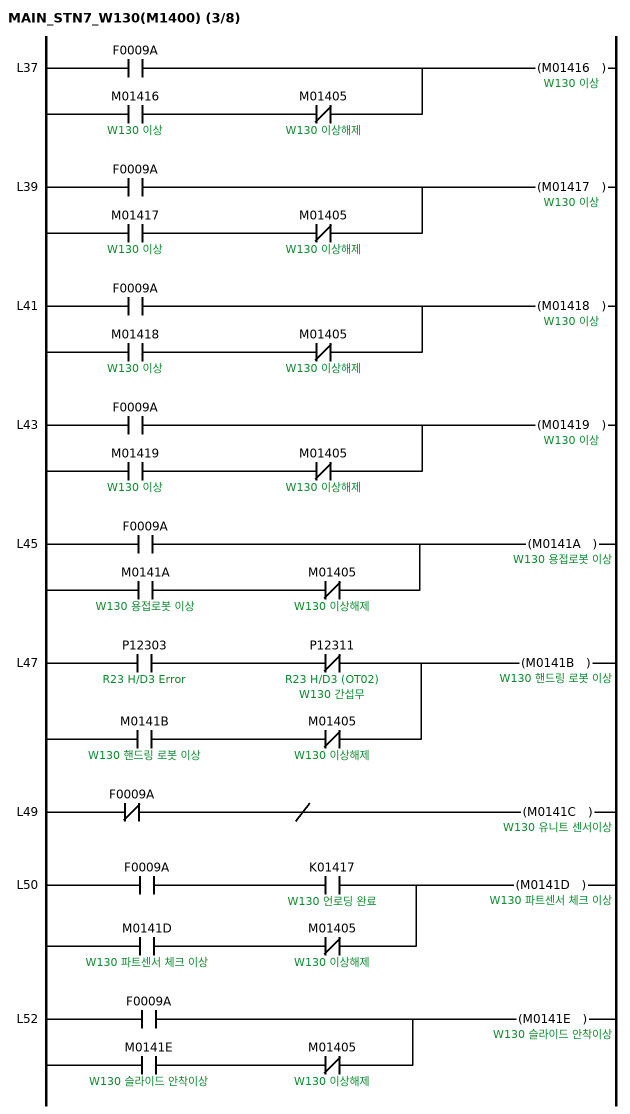
; L37
LOAD      F0009A
LOAD      M01416	// W130 이상
AND NOT   M01405	// W130 이상해제
OR LOAD
OUT       M01416	// W130 이상
; L39
LOAD      F0009A
LOAD      M01417	// W130 이상
AND NOT   M01405	// W130 이상해제
OR LOAD
OUT       M01417	// W130 이상
; L41
LOAD      F0009A
LOAD      M01418	// W130 이상
AND NOT   M01405	// W130 이상해제
OR LOAD
OUT       M01418	// W130 이상
; L43
LOAD      F0009A
LOAD      M01419	// W130 이상
AND NOT   M01405	// W130 이상해제
OR LOAD
OUT       M01419	// W130 이상
; L45
LOAD      F0009A
LOAD      M0141A	// W130 용접로봇 이상
AND NOT   M01405	// W130 이상해제
OR LOAD
OUT       M0141A	// W130 용접로봇 이상
; L47
LOAD      P12303	// R23 H/D3 Error
AND NOT   P12311	// R23 H/D3 (OT02) W130 간섭무
LOAD      M0141B	// W130 핸드링 로봇 이상
AND NOT   M01405	// W130 이상해제
OR LOAD
OUT       M0141B	// W130 핸드링 로봇 이상
; L49
LOAD NOT  F0009A
NOT
OUT       M0141C	// W130 유니트 센서이상
; L50
LOAD      F0009A
AND       K01417	// W130 언로딩 완료
LOAD      M0141D	// W130 파트센서 체크 이상
AND NOT   M01405	// W130 이상해제
OR LOAD
OUT       M0141D	// W130 파트센서 체크 이상
; L52
LOAD      F0009A
LOAD      M0141E	// W130 슬라이드 안착이상
AND NOT   M01405	// W130 이상해제
OR LOAD
OUT       M0141E	// W130 슬라이드 안착이상

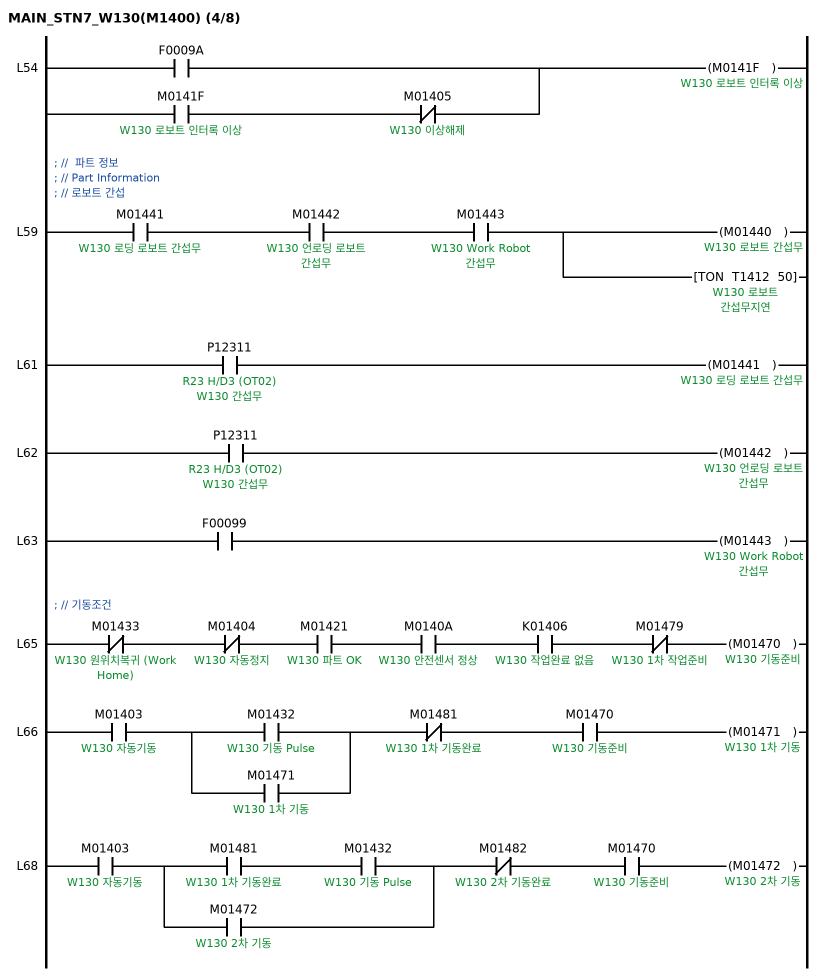
; L54
LOAD      F0009A
LOAD      M0141F	// W130 로보트 인터록 이상
AND NOT   M01405	// W130 이상해제
OR LOAD
OUT       M0141F	// W130 로보트 인터록 이상
//   //  파트 정보
//   // Part Information
//   // 로보트 간섭
; L59
LOAD      M01441	// W130 로딩 로보트 간섭무
AND       M01442	// W130 언로딩 로보트 간섭무
AND       M01443	// W130 Work Robot 간섭무
OUT       M01440	// W130 로보트 간섭무
TON       T1412 50	// W130 로보트 간섭무지연
; L61
LOAD      P12311	// R23 H/D3 (OT02) W130 간섭무
OUT       M01441	// W130 로딩 로보트 간섭무
; L62
LOAD      P12311	// R23 H/D3 (OT02) W130 간섭무
OUT       M01442	// W130 언로딩 로보트 간섭무
; L63
LOAD      F00099
OUT       M01443	// W130 Work Robot 간섭무
//   // 기동조건
; L65
LOAD NOT  M01433	// W130 원위치복귀 (Work Home)
AND NOT   M01404	// W130 자동정지
AND       M01421	// W130 파트 OK
AND       M0140A	// W130 안전센서 정상
AND       K01406	// W130 작업완료 없음
AND NOT   M01479	// W130 1차 작업준비
OUT       M01470	// W130 기동준비
; L66
LOAD      M01403	// W130 자동기동
LOAD      M01432	// W130 기동 Pulse
OR        M01471	// W130 1차 기동
AND LOAD
AND NOT   M01481	// W130 1차 기동완료
AND       M01470	// W130 기동준비
OUT       M01471	// W130 1차 기동
; L68
LOAD      M01403	// W130 자동기동
LOAD      M01481	// W130 1차 기동완료
AND       M01432	// W130 기동 Pulse
OR        M01472	// W130 2차 기동
AND LOAD
AND NOT   M01482	// W130 2차 기동완료
AND       M01470	// W130 기동준비
OUT       M01472	// W130 2차 기동

